LIN {X 0,Y 467.578,Z 154.242,A -85,B 0,C 180,E1 -7774.244,E2 -7774.244} C_VEL
LIN {X 0,Y 467.538,Z 154.245,A -85,B 0,C 180,E1 -7777.188,E2 -7777.188} C_VEL
LIN {X 0,Y 467.566,Z 154.241,A -85,B 0,C 180,E1 -7780.266,E2 -7780.266} C_VEL
LIN {X 0,Y 467.576,Z 154.241,A -85,B 0,C 180,E1 -7782.568,E2 -7782.568} C_VEL
LIN {X 0,Y 467.561,Z 154.246,A -85,B 0,C 180,E1 -7785.055,E2 -7785.055} C_VEL
LIN {X 0,Y 467.579,Z 154.241,A -85,B 0,C 180,E1 -7787.441,E2 -7787.441} C_VEL
LIN {X 0,Y 467.551,Z 154.244,A -85,B 0,C 180,E1 -7790.855,E2 -7790.855} C_VEL
LIN {X 0,Y 467.55,Z 154.243,A -85,B 0,C 180,E1 -7794.263,E2 -7794.263} C_VEL
LIN {X 0,Y 467.576,Z 154.241,A -85,B 0,C 180,E1 -7797.322,E2 -7797.322} C_VEL
LIN {X 0,Y 467.572,Z 154.242,A -85,B 0,C 180,E1 -7800.667,E2 -7800.667} C_VEL
LIN {X 0,Y 467.583,Z 154.244,A -85,B 0,C 180,E1 -7803.199,E2 -7803.199} C_VEL
LIN {X 0,Y 467.585,Z 154.242,A -85,B 0,C 180,E1 -7806.471,E2 -7806.471} C_VEL
LIN {X 0,Y 467.62,Z 154.237,A -85,B 0,C 180,E1 -7809.779,E2 -7809.779} C_VEL
LIN {X 0,Y 467.607,Z 154.238,A -85,B 0,C 180,E1 -7812.508,E2 -7812.508} C_VEL
LIN {X 0,Y 467.6,Z 154.239,A -85,B 0,C 180,E1 -7815.198,E2 -7815.198} C_VEL
LIN {X 0,Y 467.59,Z 154.239,A -85,B 0,C 180,E1 -7815.443,E2 -7815.443} C_VEL
LIN {X 0,Y 466.92,Z 154.324,A -85,B 0,C 180,E1 -7816.162,E2 -7816.162} C_VEL
LIN {X 0,Y 464.077,Z 154.675,A -85,B 0,C 180,E1 -7817.33,E2 -7817.33} C_VEL
LIN {X 0,Y 461.679,Z 154.979,A -85,B 0,C 180,E1 -7818.273,E2 -7818.273} C_VEL
LIN {X 0,Y 460.653,Z 155.102,A -85,B 0,C 180,E1 -7819,E2 -7819} C_VEL
LIN {X 0,Y 460.571,Z 155.112,A -85,B 0,C 180,E1 -7819.247,E2 -7819.247} C_VEL
LIN {X 0,Y 460.721,Z 155.095,A -85,B 0,C 180,E1 -7822.54,E2 -7822.54} C_VEL
LIN {X 0,Y 460.698,Z 155.101,A -85,B 0,C 180,E1 -7824.75,E2 -7824.75} C_VEL
LIN {X 0,Y 460.801,Z 155.085,A -85,B 0,C 180,E1 -7827.379,E2 -7827.379} C_VEL
LIN {X 0,Y 460.821,Z 155.086,A -85,B 0,C 180,E1 -7830.001,E2 -7830.001} C_VEL
LIN {X 0,Y 460.793,Z 155.085,A -85,B 0,C 180,E1 -7832.624,E2 -7832.624} C_VEL
LIN {X 0,Y 460.713,Z 155.097,A -85,B 0,C 180,E1 -7836.131,E2 -7836.131} C_VEL
LIN {X 0,Y 460.63,Z 155.107,A -85,B 0,C 180,E1 -7838.777,E2 -7838.777} C_VEL
LIN {X 0,Y 460.6,Z 155.109,A -85,B 0,C 180,E1 -7842.436,E2 -7842.436} C_VEL
LIN {X 0,Y 460.605,Z 155.109,A -85,B 0,C 180,E1 -7845.999,E2 -7845.999} C_VEL
LIN {X 0,Y 460.573,Z 155.114,A -85,B 0,C 180,E1 -7849.617,E2 -7849.617} C_VEL
LIN {X 0,Y 460.515,Z 155.122,A -85,B 0,C 180,E1 -7852.43,E2 -7852.43} C_VEL
LIN {X 0,Y 460.538,Z 155.116,A -85,B 0,C 180,E1 -7855.794,E2 -7855.794} C_VEL
LIN {X 0,Y 460.525,Z 155.12,A -85,B 0,C 180,E1 -7859.233,E2 -7859.233} C_VEL
LIN {X 0,Y 460.534,Z 155.121,A -85,B 0,C 180,E1 -7862.285,E2 -7862.285} C_VEL
LIN {X 0,Y 460.51,Z 155.123,A -85,B 0,C 180,E1 -7865.447,E2 -7865.447} C_VEL
LIN {X 0,Y 460.495,Z 155.125,A -85,B 0,C 180,E1 -7868.89,E2 -7868.89} C_VEL
LIN {X 0,Y 460.514,Z 155.121,A -85,B 0,C 180,E1 -7871.6,E2 -7871.6} C_VEL
LIN {X 0,Y 460.517,Z 155.121,A -85,B 0,C 180,E1 -7874.59,E2 -7874.59} C_VEL
LIN {X 0,Y 460.528,Z 155.119,A -85,B 0,C 180,E1 -7877.819,E2 -7877.819} C_VEL
LIN {X 0,Y 460.526,Z 155.12,A -85,B 0,C 180,E1 -7880.137,E2 -7880.137} C_VEL
LIN {X 0,Y 460.47,Z 155.126,A -85,B 0,C 180,E1 -7883.47,E2 -7883.47} C_VEL
LIN {X 0,Y 460.529,Z 155.12,A -85,B 0,C 180,E1 -7886.675,E2 -7886.675} C_VEL
LIN {X 0,Y 460.61,Z 155.131,A -85,B 0,C 180,E1 -7887.845,E2 -7887.845} C_VEL
LIN {X 0,Y 461.333,Z 159.923,A -85,B 0,C 180,E1 -7889.82,E2 -7889.82} C_VEL
LIN {X 0,Y 461.056,Z 167.48,A -85,B 0,C 180,E1 -7892.787,E2 -7892.787} C_VEL
LIN {X 0,Y 460.72,Z 176.433,A -85,B 0,C 180,E1 -7896.245,E2 -7896.245} C_VEL
LIN {X 0,Y 460.469,Z 184.873,A -85,B 0,C 180,E1 -7899.449,E2 -7899.449} C_VEL
LIN {X 0,Y 460.238,Z 193.485,A -85,B 0,C 180,E1 -7902.676,E2 -7902.676} C_VEL
LIN {X 0,Y 460.05,Z 202.076,A -85,B 0,C 180,E1 -7905.852,E2 -7905.852} C_VEL
LIN {X 0,Y 459.9,Z 210.667,A -85,B 0,C 180,E1 -7908.988,E2 -7908.988} C_VEL
LIN {X 0,Y 459.815,Z 215.225,A -85,B 0,C 180,E1 -7910.599,E2 -7910.599} C_VEL
LIN {X 0,Y 460.939,Z 225.296,A -85,B 0,C 180,E1 -7911.064,E2 -7911.064} C_VEL
LIN {X 0,Y 461.025,Z 231.865,A -85,B 0,C 180,E1 -7911.452,E2 -7911.452} C_VEL
LIN {X 0,Y 460.704,Z 240.677,A -85,B 0,C 180,E1 -7912.109,E2 -7912.109} C_VEL
LIN {X 0,Y 460.448,Z 249.624,A -85,B 0,C 180,E1 -7912.986,E2 -7912.986} C_VEL
LIN {X 0,Y 460.224,Z 256.55,A -85,B 0,C 180,E1 -7913.864,E2 -7913.864} C_VEL
LIN {X 0,Y 460.116,Z 263.238,A -85,B 0,C 180,E1 -7914.961,E2 -7914.961} C_VEL
LIN {X 0,Y 459.946,Z 268.255,A -85,B 0,C 180,E1 -7916.057,E2 -7916.057} C_VEL
LIN {X 0,Y 459.732,Z 272.503,A -85,B 0,C 180,E1 -7917.371,E2 -7917.371} C_VEL
LIN {X 0,Y 459.652,Z 274.384,A -85,B 0,C 180,E1 -7918.248,E2 -7918.248} C_VEL
LIN {X 0,Y 459.577,Z 275.564,A -85,B 0,C 180,E1 -7919.124,E2 -7919.124} C_VEL
LIN {X 0,Y 459.558,Z 276.065,A -85,B 0,C 180,E1 -7920,E2 -7920} C_VEL
LIN {X 0,Y 459.579,Z 275.892,A -85,B 0,C 180,E1 -7920.876,E2 -7920.876} C_VEL
LIN {X 0,Y 459.655,Z 275.048,A -85,B 0,C 180,E1 -7921.752,E2 -7921.752} C_VEL
LIN {X 0,Y 459.875,Z 272.488,A -85,B 0,C 180,E1 -7923.066,E2 -7923.066} C_VEL
LIN {X 0,Y 460.05,Z 269.86,A -85,B 0,C 180,E1 -7923.942,E2 -7923.942} C_VEL
LIN {X 0,Y 460.191,Z 265.403,A -85,B 0,C 180,E1 -7925.038,E2 -7925.038} C_VEL
LIN {X 0,Y 460.275,Z 259.447,A -85,B 0,C 180,E1 -7926.136,E2 -7926.136} C_VEL
LIN {X 0,Y 460.601,Z 252.231,A -85,B 0,C 180,E1 -7927.147,E2 -7927.147} C_VEL
LIN {X 0,Y 461.059,Z 243.259,A -85,B 0,C 180,E1 -7928.106,E2 -7928.106} C_VEL
LIN {X 0,Y 461.405,Z 235.329,A -85,B 0,C 180,E1 -7928.761,E2 -7928.761} C_VEL
LIN {X 0,Y 461.515,Z 226.898,A -85,B 0,C 180,E1 -7929.311,E2 -7929.311} C_VEL
LIN {X 0,Y 460.127,Z 217.109,A -85,B 0,C 180,E1 -7929.839,E2 -7929.839} C_VEL
LIN {X 0,Y 459.966,Z 215.738,A -85,B 0,C 180,E1 -7929.926,E2 -7929.926} C_VEL
LIN {X 0,Y 460.14,Z 208.06,A -85,B 0,C 180,E1 -7932.795,E2 -7932.795} C_VEL
LIN {X 0,Y 460.413,Z 199.745,A -85,B 0,C 180,E1 -7935.948,E2 -7935.948} C_VEL
LIN {X 0,Y 460.666,Z 192.048,A -85,B 0,C 180,E1 -7938.934,E2 -7938.934} C_VEL
LIN {X 0,Y 460.956,Z 184.495,A -85,B 0,C 180,E1 -7941.934,E2 -7941.934} C_VEL
LIN {X 0,Y 461.333,Z 176.432,A -85,B 0,C 180,E1 -7945.249,E2 -7945.249} C_VEL
LIN {X 0,Y 461.894,Z 169.657,A -85,B 0,C 180,E1 -7948.144,E2 -7948.144} C_VEL
LIN {X 0,Y 462.207,Z 164.213,A -85,B 0,C 180,E1 -7950.623,E2 -7950.623} C_VEL
LIN {X 0,Y 461.444,Z 159.416,A -85,B 0,C 180,E1 -7953.103,E2 -7953.103} C_VEL
LIN {X 0,Y 460.528,Z 155.123,A -85,B 0,C 180,E1 -7955.656,E2 -7955.656} C_VEL
LIN {X 0,Y 460.55,Z 155.12,A -85,B 0,C 180,E1 -7958.897,E2 -7958.897} C_VEL
LIN {X 0,Y 460.529,Z 155.122,A -85,B 0,C 180,E1 -7962.181,E2 -7962.181} C_VEL
LIN {X 0,Y 460.52,Z 155.123,A -85,B 0,C 180,E1 -7965.411,E2 -7965.411} C_VEL
LIN {X 0,Y 460.538,Z 155.12,A -85,B 0,C 180,E1 -7968.397,E2 -7968.397} C_VEL
LIN {X 0,Y 460.532,Z 155.122,A -85,B 0,C 180,E1 -7971.266,E2 -7971.266} C_VEL
LIN {X 0,Y 460.514,Z 155.125,A -85,B 0,C 180,E1 -7974.554,E2 -7974.554} C_VEL
LIN {X 0,Y 460.536,Z 155.127,A -85,B 0,C 180,E1 -7975.256,E2 -7975.256} C_VEL
LIN {X 0,Y 461.79,Z 160.451,A -85,B 0,C 180,E1 -7977.813,E2 -7977.813} C_VEL
LIN {X 0,Y 463.204,Z 167.084,A -85,B 0,C 180,E1 -7980.454,E2 -7980.454} C_VEL
LIN {X 0,Y 463.988,Z 171.493,A -85,B 0,C 180,E1 -7981.993,E2 -7981.993} C_VEL
LIN {X 0,Y 463.796,Z 176.053,A -85,B 0,C 180,E1 -7983.386,E2 -7983.386} C_VEL
LIN {X 0,Y 462.66,Z 186.329,A -85,B 0,C 180,E1 -7986.261,E2 -7986.261} C_VEL
LIN {X 0,Y 461.697,Z 198.798,A -85,B 0,C 180,E1 -7989.505,E2 -7989.505} C_VEL
LIN {X 0,Y 461.026,Z 209.902,A -85,B 0,C 180,E1 -7992.248,E2 -7992.248} C_VEL
LIN {X 0,Y 460.564,Z 220.479,A -85,B 0,C 180,E1 -7994.765,E2 -7994.765} C_VEL
LIN {X 0,Y 462.121,Z 233.34,A -85,B 0,C 180,E1 -7995.17,E2 -7995.17} C_VEL
LIN {X 0,Y 462.47,Z 239.24,A -85,B 0,C 180,E1 -7995.393,E2 -7995.393} C_VEL
LIN {X 0,Y 462.083,Z 251.878,A -85,B 0,C 180,E1 -7995.971,E2 -7995.971} C_VEL
LIN {X 0,Y 461.634,Z 263.462,A -85,B 0,C 180,E1 -7996.686,E2 -7996.686} C_VEL
LIN {X 0,Y 461.188,Z 274.136,A -85,B 0,C 180,E1 -7997.522,E2 -7997.522} C_VEL
LIN {X 0,Y 460.843,Z 283.737,A -85,B 0,C 180,E1 -7998.452,E2 -7998.452} C_VEL
LIN {X 0,Y 460.356,Z 293.826,A -85,B 0,C 180,E1 -7999.665,E2 -7999.665} C_VEL
LIN {X 0,Y 460.039,Z 302.681,A -85,B 0,C 180,E1 -8000.99,E2 -8000.99} C_VEL
LIN {X 0,Y 459.842,Z 309.702,A -85,B 0,C 180,E1 -8002.313,E2 -8002.313} C_VEL
LIN {X 0,Y 459.656,Z 316.123,A -85,B 0,C 180,E1 -8003.855,E2 -8003.855} C_VEL
LIN {X 0,Y 459.628,Z 320.303,A -85,B 0,C 180,E1 -8005.174,E2 -8005.174} C_VEL
LIN {X 0,Y 459.628,Z 323.383,A -85,B 0,C 180,E1 -8006.492,E2 -8006.492} C_VEL
LIN {X 0,Y 459.622,Z 324.86,A -85,B 0,C 180,E1 -8007.369,E2 -8007.369} C_VEL
LIN {X 0,Y 459.601,Z 325.903,A -85,B 0,C 180,E1 -8008.246,E2 -8008.246} C_VEL
LIN {X 0,Y 459.56,Z 326.544,A -85,B 0,C 180,E1 -8009.122,E2 -8009.122} C_VEL
LIN {X 0,Y 459.542,Z 326.768,A -85,B 0,C 180,E1 -8009.999,E2 -8009.999} C_VEL
LIN {X 0,Y 459.63,Z 325.922,A -85,B 0,C 180,E1 -8011.751,E2 -8011.751} C_VEL
LIN {X 0,Y 459.621,Z 324.894,A -85,B 0,C 180,E1 -8012.628,E2 -8012.628} C_VEL
LIN {X 0,Y 459.641,Z 323.396,A -85,B 0,C 180,E1 -8013.505,E2 -8013.505} C_VEL
LIN {X 0,Y 459.623,Z 320.313,A -85,B 0,C 180,E1 -8014.823,E2 -8014.823} C_VEL
LIN {X 0,Y 459.713,Z 315.065,A -85,B 0,C 180,E1 -8016.429,E2 -8016.429} C_VEL
LIN {X 0,Y 459.866,Z 308.616,A -85,B 0,C 180,E1 -8017.904,E2 -8017.904} C_VEL
LIN {X 0,Y 460.097,Z 301.234,A -85,B 0,C 180,E1 -8019.228,E2 -8019.228} C_VEL
LIN {X 0,Y 460.348,Z 293.675,A -85,B 0,C 180,E1 -8020.332,E2 -8020.332} C_VEL
LIN {X 0,Y 460.797,Z 284.488,A -85,B 0,C 180,E1 -8021.434,E2 -8021.434} C_VEL
LIN {X 0,Y 461.196,Z 274.181,A -85,B 0,C 180,E1 -8022.43,E2 -8022.43} C_VEL
LIN {X 0,Y 461.628,Z 262.754,A -85,B 0,C 180,E1 -8023.311,E2 -8023.311} C_VEL
LIN {X 0,Y 462.054,Z 250.719,A -85,B 0,C 180,E1 -8024.027,E2 -8024.027} C_VEL
LIN {X 0,Y 462.432,Z 237.387,A -85,B 0,C 180,E1 -8024.606,E2 -8024.606} C_VEL
LIN {X 0,Y 460.969,Z 224.354,A -85,B 0,C 180,E1 -8025.02,E2 -8025.02} C_VEL
LIN {X 0,Y 460.482,Z 220.513,A -85,B 0,C 180,E1 -8025.121,E2 -8025.121} C_VEL
LIN {X 0,Y 461.162,Z 205.323,A -85,B 0,C 180,E1 -8028.663,E2 -8028.663} C_VEL
LIN {X 0,Y 461.925,Z 189.777,A -85,B 0,C 180,E1 -8032.354,E2 -8032.354} C_VEL
LIN {X 0,Y 462.774,Z 176.253,A -85,B 0,C 180,E1 -8035.645,E2 -8035.645} C_VEL
LIN {X 0,Y 463.153,Z 170.459,A -85,B 0,C 180,E1 -8037.078,E2 -8037.078} C_VEL
LIN {X 0,Y 462.725,Z 165.962,A -85,B 0,C 180,E1 -8038.246,E2 -8038.246} C_VEL
LIN {X 0,Y 460.54,Z 155.121,A -85,B 0,C 180,E1 -8041.227,E2 -8041.227} C_VEL
LIN {X 0,Y 460.529,Z 155.122,A -85,B 0,C 180,E1 -8044.504,E2 -8044.504} C_VEL
LIN {X 0,Y 460.521,Z 155.121,A -85,B 0,C 180,E1 -8047.619,E2 -8047.619} C_VEL
LIN {X 0,Y 460.518,Z 155.121,A -85,B 0,C 180,E1 -8051.01,E2 -8051.01} C_VEL
LIN {X 0,Y 460.506,Z 155.123,A -85,B 0,C 180,E1 -8054.587,E2 -8054.587} C_VEL
LIN {X 0,Y 460.538,Z 155.12,A -85,B 0,C 180,E1 -8057.82,E2 -8057.82} C_VEL
LIN {X 0,Y 460.557,Z 155.116,A -85,B 0,C 180,E1 -8061.097,E2 -8061.097} C_VEL
LIN {X 0,Y 460.496,Z 155.123,A -85,B 0,C 180,E1 -8064.553,E2 -8064.553} C_VEL
LIN {X 0,Y 460.521,Z 155.123,A -85,B 0,C 180,E1 -8067.715,E2 -8067.715} C_VEL
LIN {X 0,Y 460.535,Z 155.12,A -85,B 0,C 180,E1 -8070.769,E2 -8070.769} C_VEL
LIN {X 0,Y 460.551,Z 155.117,A -85,B 0,C 180,E1 -8073.734,E2 -8073.734} C_VEL
LIN {X 0,Y 460.531,Z 155.117,A -85,B 0,C 180,E1 -8076.623,E2 -8076.623} C_VEL
LIN {X 0,Y 460.537,Z 155.122,A -85,B 0,C 180,E1 -8079.452,E2 -8079.452} C_VEL
LIN {X 0,Y 460.546,Z 155.118,A -85,B 0,C 180,E1 -8082.229,E2 -8082.229} C_VEL
LIN {X 0,Y 460.551,Z 155.117,A -85,B 0,C 180,E1 -8084.964,E2 -8084.964} C_VEL
LIN {X 0,Y 460.613,Z 155.112,A -85,B 0,C 180,E1 -8087.666,E2 -8087.666} C_VEL
LIN {X 0,Y 460.611,Z 155.112,A -85,B 0,C 180,E1 -8091.223,E2 -8091.223} C_VEL
LIN {X 0,Y 460.698,Z 155.098,A -85,B 0,C 180,E1 -8093.87,E2 -8093.87} C_VEL
LIN {X 0,Y 460.812,Z 155.086,A -85,B 0,C 180,E1 -8097.378,E2 -8097.378} C_VEL
LIN {X 0,Y 460.836,Z 155.081,A -85,B 0,C 180,E1 -8100,E2 -8100} C_VEL
LIN {X 0,Y 460.78,Z 155.089,A -85,B 0,C 180,E1 -8102.623,E2 -8102.623} C_VEL
LIN {X 0,Y 460.694,Z 155.1,A -85,B 0,C 180,E1 -8106.13,E2 -8106.13} C_VEL
LIN {X 0,Y 460.615,Z 155.109,A -85,B 0,C 180,E1 -8108.776,E2 -8108.776} C_VEL
LIN {X 0,Y 460.619,Z 155.109,A -85,B 0,C 180,E1 -8112.457,E2 -8112.457} C_VEL
LIN {X 0,Y 460.585,Z 155.112,A -85,B 0,C 180,E1 -8115.998,E2 -8115.998} C_VEL
LIN {X 0,Y 460.557,Z 155.116,A -85,B 0,C 180,E1 -8118.903,E2 -8118.903} C_VEL
LIN {X 0,Y 460.549,Z 155.118,A -85,B 0,C 180,E1 -8121.484,E2 -8121.484} C_VEL
LIN {X 0,Y 460.524,Z 155.122,A -85,B 0,C 180,E1 -8124.333,E2 -8124.333} C_VEL
LIN {X 0,Y 460.521,Z 155.118,A -85,B 0,C 180,E1 -8127.247,E2 -8127.247} C_VEL
LIN {X 0,Y 460.496,Z 155.123,A -85,B 0,C 180,E1 -8130.241,E2 -8130.241} C_VEL
LIN {X 0,Y 460.517,Z 155.123,A -85,B 0,C 180,E1 -8133.326,E2 -8133.326} C_VEL
LIN {X 0,Y 460.467,Z 155.128,A -85,B 0,C 180,E1 -8136.53,E2 -8136.53} C_VEL
LIN {X 0,Y 460.546,Z 155.119,A -85,B 0,C 180,E1 -8139.861,E2 -8139.861} C_VEL
LIN {X 0,Y 460.506,Z 155.122,A -85,B 0,C 180,E1 -8142.902,E2 -8142.902} C_VEL
LIN {X 0,Y 460.51,Z 155.122,A -85,B 0,C 180,E1 -8145.831,E2 -8145.831} C_VEL
LIN {X 0,Y 460.524,Z 155.12,A -85,B 0,C 180,E1 -8148.99,E2 -8148.99} C_VEL
LIN {X 0,Y 460.51,Z 155.124,A -85,B 0,C 180,E1 -8151.268,E2 -8151.268} C_VEL
LIN {X 0,Y 460.501,Z 155.122,A -85,B 0,C 180,E1 -8154.556,E2 -8154.556} C_VEL
LIN {X 0,Y 460.527,Z 155.12,A -85,B 0,C 180,E1 -8157.717,E2 -8157.717} C_VEL
LIN {X 0,Y 460.541,Z 155.118,A -85,B 0,C 180,E1 -8160.771,E2 -8160.771} C_VEL
LIN {X 0,Y 460.537,Z 155.117,A -85,B 0,C 180,E1 -8163.735,E2 -8163.735} C_VEL
LIN {X 0,Y 460.539,Z 155.121,A -85,B 0,C 180,E1 -8166.625,E2 -8166.625} C_VEL
LIN {X 0,Y 460.548,Z 155.117,A -85,B 0,C 180,E1 -8169.454,E2 -8169.454} C_VEL
LIN {X 0,Y 460.557,Z 155.116,A -85,B 0,C 180,E1 -8172.232,E2 -8172.232} C_VEL
LIN {X 0,Y 460.56,Z 155.117,A -85,B 0,C 180,E1 -8174.966,E2 -8174.966} C_VEL
LIN {X 0,Y 460.608,Z 155.111,A -85,B 0,C 180,E1 -8178.561,E2 -8178.561} C_VEL
LIN {X 0,Y 460.571,Z 155.112,A -85,B 0,C 180,E1 -8179.247,E2 -8179.247} C_VEL
LIN {X 0,Y 459.917,Z 155.198,A -85,B 0,C 180,E1 -8179.977,E2 -8179.977} C_VEL
LIN {X 0,Y 457.101,Z 155.547,A -85,B 0,C 180,E1 -8181.164,E2 -8181.164} C_VEL
LIN {X 0,Y 454.725,Z 155.844,A -85,B 0,C 180,E1 -8182.121,E2 -8182.121} C_VEL
LIN {X 0,Y 453.715,Z 155.969,A -85,B 0,C 180,E1 -8182.86,E2 -8182.86} C_VEL
LIN {X 0,Y 453.638,Z 155.978,A -85,B 0,C 180,E1 -8183.11,E2 -8183.11} C_VEL
LIN {X 0,Y 453.672,Z 155.975,A -85,B 0,C 180,E1 -8184.668,E2 -8184.668} C_VEL
LIN {X 0,Y 453.746,Z 155.964,A -85,B 0,C 180,E1 -8187.338,E2 -8187.338} C_VEL
LIN {X 0,Y 453.79,Z 155.962,A -85,B 0,C 180,E1 -8190.001,E2 -8190.001} C_VEL
LIN {X 0,Y 453.737,Z 155.964,A -85,B 0,C 180,E1 -8192.665,E2 -8192.665} C_VEL
LIN {X 0,Y 453.68,Z 155.973,A -85,B 0,C 180,E1 -8196.227,E2 -8196.227} C_VEL
LIN {X 0,Y 453.594,Z 155.984,A -85,B 0,C 180,E1 -8198.915,E2 -8198.915} C_VEL
LIN {X 0,Y 453.567,Z 155.985,A -85,B 0,C 180,E1 -8202.53,E2 -8202.53} C_VEL
LIN {X 0,Y 453.549,Z 155.988,A -85,B 0,C 180,E1 -8206.197,E2 -8206.197} C_VEL
LIN {X 0,Y 453.522,Z 155.994,A -85,B 0,C 180,E1 -8209.041,E2 -8209.041} C_VEL
LIN {X 0,Y 453.481,Z 155.999,A -85,B 0,C 180,E1 -8211.837,E2 -8211.837} C_VEL
LIN {X 0,Y 453.473,Z 155.997,A -85,B 0,C 180,E1 -8214.738,E2 -8214.738} C_VEL
LIN {X 0,Y 453.467,Z 155.998,A -85,B 0,C 180,E1 -8217.944,E2 -8217.944} C_VEL
LIN {X 0,Y 453.479,Z 155.999,A -85,B 0,C 180,E1 -8220.761,E2 -8220.761} C_VEL
LIN {X 0,Y 453.473,Z 155.999,A -85,B 0,C 180,E1 -8223.914,E2 -8223.914} C_VEL
LIN {X 0,Y 453.443,Z 156.003,A -85,B 0,C 180,E1 -8227.192,E2 -8227.192} C_VEL
LIN {X 0,Y 453.475,Z 156,A -85,B 0,C 180,E1 -8230.612,E2 -8230.612} C_VEL
LIN {X 0,Y 453.465,Z 156.001,A -85,B 0,C 180,E1 -8234.222,E2 -8234.222} C_VEL
LIN {X 0,Y 453.467,Z 156.001,A -85,B 0,C 180,E1 -8237.005,E2 -8237.005} C_VEL
LIN {X 0,Y 453.499,Z 155.994,A -85,B 0,C 180,E1 -8239.41,E2 -8239.41} C_VEL
LIN {X 0,Y 453.444,Z 156.001,A -85,B 0,C 180,E1 -8242.809,E2 -8242.809} C_VEL
LIN {X 0,Y 453.475,Z 155.999,A -85,B 0,C 180,E1 -8246.087,E2 -8246.087} C_VEL
LIN {X 0,Y 453.588,Z 156.076,A -85,B 0,C 180,E1 -8247.752,E2 -8247.752} C_VEL
LIN {X 0,Y 454.308,Z 161.581,A -85,B 0,C 180,E1 -8250.033,E2 -8250.033} C_VEL
LIN {X 0,Y 453.974,Z 169.864,A -85,B 0,C 180,E1 -8253.324,E2 -8253.324} C_VEL
LIN {X 0,Y 453.622,Z 178.6,A -85,B 0,C 180,E1 -8256.729,E2 -8256.729} C_VEL
LIN {X 0,Y 453.381,Z 187.277,A -85,B 0,C 180,E1 -8260.06,E2 -8260.06} C_VEL
LIN {X 0,Y 453.168,Z 195.94,A -85,B 0,C 180,E1 -8263.327,E2 -8263.327} C_VEL
LIN {X 0,Y 452.947,Z 204.557,A -85,B 0,C 180,E1 -8266.541,E2 -8266.541} C_VEL
LIN {X 0,Y 452.762,Z 213.16,A -85,B 0,C 180,E1 -8269.717,E2 -8269.717} C_VEL
LIN {X 0,Y 452.753,Z 215.324,A -85,B 0,C 180,E1 -8270.451,E2 -8270.451} C_VEL
LIN {X 0,Y 453.895,Z 225.363,A -85,B 0,C 180,E1 -8270.924,E2 -8270.924} C_VEL
LIN {X 0,Y 454.018,Z 231.934,A -85,B 0,C 180,E1 -8271.319,E2 -8271.319} C_VEL
LIN {X 0,Y 453.675,Z 240.772,A -85,B 0,C 180,E1 -8271.986,E2 -8271.986} C_VEL
LIN {X 0,Y 453.405,Z 249.758,A -85,B 0,C 180,E1 -8272.877,E2 -8272.877} C_VEL
LIN {X 0,Y 453.184,Z 256.726,A -85,B 0,C 180,E1 -8273.768,E2 -8273.768} C_VEL
LIN {X 0,Y 453.038,Z 263.457,A -85,B 0,C 180,E1 -8274.882,E2 -8274.882} C_VEL
LIN {X 0,Y 452.88,Z 268.517,A -85,B 0,C 180,E1 -8275.996,E2 -8275.996} C_VEL
LIN {X 0,Y 452.656,Z 272.809,A -85,B 0,C 180,E1 -8277.33,E2 -8277.33} C_VEL
LIN {X 0,Y 452.576,Z 274.721,A -85,B 0,C 180,E1 -8278.22,E2 -8278.22} C_VEL
LIN {X 0,Y 452.512,Z 275.932,A -85,B 0,C 180,E1 -8279.11,E2 -8279.11} C_VEL
LIN {X 0,Y 452.491,Z 276.463,A -85,B 0,C 180,E1 -8280,E2 -8280} C_VEL
LIN {X 0,Y 452.513,Z 276.322,A -85,B 0,C 180,E1 -8280.89,E2 -8280.89} C_VEL
LIN {X 0,Y 452.596,Z 275.507,A -85,B 0,C 180,E1 -8281.78,E2 -8281.78} C_VEL
LIN {X 0,Y 452.828,Z 272.992,A -85,B 0,C 180,E1 -8283.114,E2 -8283.114} C_VEL
LIN {X 0,Y 453.005,Z 270.405,A -85,B 0,C 180,E1 -8284.003,E2 -8284.003} C_VEL
LIN {X 0,Y 453.159,Z 266.01,A -85,B 0,C 180,E1 -8285.116,E2 -8285.116} C_VEL
LIN {X 0,Y 453.254,Z 260.142,A -85,B 0,C 180,E1 -8286.231,E2 -8286.231} C_VEL
LIN {X 0,Y 453.627,Z 253.039,A -85,B 0,C 180,E1 -8287.257,E2 -8287.257} C_VEL
LIN {X 0,Y 454.099,Z 244.254,A -85,B 0,C 180,E1 -8288.231,E2 -8288.231} C_VEL
LIN {X 0,Y 454.541,Z 235.084,A -85,B 0,C 180,E1 -8289.007,E2 -8289.007} C_VEL
LIN {X 0,Y 454.536,Z 226.624,A -85,B 0,C 180,E1 -8289.568,E2 -8289.568} C_VEL
LIN {X 0,Y 452.893,Z 215.887,A -85,B 0,C 180,E1 -8290.167,E2 -8290.167} C_VEL
LIN {X 0,Y 453.11,Z 208.424,A -85,B 0,C 180,E1 -8292.997,E2 -8292.997} C_VEL
LIN {X 0,Y 453.415,Z 200.124,A -85,B 0,C 180,E1 -8296.201,E2 -8296.201} C_VEL
LIN {X 0,Y 453.711,Z 192.031,A -85,B 0,C 180,E1 -8299.406,E2 -8299.406} C_VEL
LIN {X 0,Y 453.987,Z 184.947,A -85,B 0,C 180,E1 -8302.289,E2 -8302.289} C_VEL
LIN {X 0,Y 454.387,Z 178.087,A -85,B 0,C 180,E1 -8305.172,E2 -8305.172} C_VEL
LIN {X 0,Y 455.015,Z 170.966,A -85,B 0,C 180,E1 -8308.308,E2 -8308.308} C_VEL
LIN {X 0,Y 455.326,Z 165.982,A -85,B 0,C 180,E1 -8310.621,E2 -8310.621} C_VEL
LIN {X 0,Y 454.732,Z 161.992,A -85,B 0,C 180,E1 -8312.747,E2 -8312.747} C_VEL
LIN {X 0,Y 453.987,Z 158.278,A -85,B 0,C 180,E1 -8314.945,E2 -8314.945} C_VEL
LIN {X 0,Y 453.45,Z 156.005,A -85,B 0,C 180,E1 -8316.583,E2 -8316.583} C_VEL
LIN {X 0,Y 453.496,Z 155.999,A -85,B 0,C 180,E1 -8319.449,E2 -8319.449} C_VEL
LIN {X 0,Y 453.482,Z 155.999,A -85,B 0,C 180,E1 -8321.934,E2 -8321.934} C_VEL
LIN {X 0,Y 453.491,Z 155.998,A -85,B 0,C 180,E1 -8325.471,E2 -8325.471} C_VEL
LIN {X 0,Y 453.485,Z 155.999,A -85,B 0,C 180,E1 -8328.209,E2 -8328.209} C_VEL
LIN {X 0,Y 453.5,Z 155.998,A -85,B 0,C 180,E1 -8330.793,E2 -8330.793} C_VEL
LIN {X 0,Y 453.478,Z 156.021,A -85,B 0,C 180,E1 -8334.329,E2 -8334.329} C_VEL
LIN {X 0,Y 454.505,Z 160.218,A -85,B 0,C 180,E1 -8336.616,E2 -8336.616} C_VEL
LIN {X 0,Y 455.912,Z 166.574,A -85,B 0,C 180,E1 -8339.421,E2 -8339.421} C_VEL
LIN {X 0,Y 457.004,Z 172.24,A -85,B 0,C 180,E1 -8341.527,E2 -8341.527} C_VEL
LIN {X 0,Y 457.184,Z 175.23,A -85,B 0,C 180,E1 -8342.536,E2 -8342.536} C_VEL
LIN {X 0,Y 456.05,Z 185.023,A -85,B 0,C 180,E1 -8345.411,E2 -8345.411} C_VEL
LIN {X 0,Y 454.888,Z 197.193,A -85,B 0,C 180,E1 -8348.71,E2 -8348.71} C_VEL
LIN {X 0,Y 454.07,Z 209.97,A -85,B 0,C 180,E1 -8351.966,E2 -8351.966} C_VEL
LIN {X 0,Y 453.56,Z 220.544,A -85,B 0,C 180,E1 -8354.537,E2 -8354.537} C_VEL
LIN {X 0,Y 455.114,Z 232.788,A -85,B 0,C 180,E1 -8354.922,E2 -8354.922} C_VEL
LIN {X 0,Y 455.569,Z 239.804,A -85,B 0,C 180,E1 -8355.195,E2 -8355.195} C_VEL
LIN {X 0,Y 455.183,Z 251.645,A -85,B 0,C 180,E1 -8355.753,E2 -8355.753} C_VEL
LIN {X 0,Y 454.706,Z 263.183,A -85,B 0,C 180,E1 -8356.479,E2 -8356.479} C_VEL
LIN {X 0,Y 454.186,Z 274.366,A -85,B 0,C 180,E1 -8357.374,E2 -8357.374} C_VEL
LIN {X 0,Y 453.805,Z 284.42,A -85,B 0,C 180,E1 -8358.384,E2 -8358.384} C_VEL
LIN {X 0,Y 453.34,Z 293.498,A -85,B 0,C 180,E1 -8359.503,E2 -8359.503} C_VEL
LIN {X 0,Y 452.993,Z 302.337,A -85,B 0,C 180,E1 -8360.848,E2 -8360.848} C_VEL
LIN {X 0,Y 452.757,Z 309.345,A -85,B 0,C 180,E1 -8362.192,E2 -8362.192} C_VEL
LIN {X 0,Y 452.585,Z 315.769,A -85,B 0,C 180,E1 -8363.758,E2 -8363.758} C_VEL
LIN {X 0,Y 452.558,Z 319.943,A -85,B 0,C 180,E1 -8365.099,E2 -8365.099} C_VEL
LIN {X 0,Y 452.525,Z 323.013,A -85,B 0,C 180,E1 -8366.437,E2 -8366.437} C_VEL
LIN {X 0,Y 452.544,Z 324.483,A -85,B 0,C 180,E1 -8367.328,E2 -8367.328} C_VEL
LIN {X 0,Y 452.511,Z 325.521,A -85,B 0,C 180,E1 -8368.219,E2 -8368.219} C_VEL
LIN {X 0,Y 452.495,Z 326.159,A -85,B 0,C 180,E1 -8369.109,E2 -8369.109} C_VEL
LIN {X 0,Y 452.475,Z 326.369,A -85,B 0,C 180,E1 -8369.999,E2 -8369.999} C_VEL
LIN {X 0,Y 452.495,Z 326.137,A -85,B 0,C 180,E1 -8370.889,E2 -8370.889} C_VEL
LIN {X 0,Y 452.538,Z 325.507,A -85,B 0,C 180,E1 -8371.778,E2 -8371.778} C_VEL
LIN {X 0,Y 452.544,Z 324.467,A -85,B 0,C 180,E1 -8372.669,E2 -8372.669} C_VEL
LIN {X 0,Y 452.539,Z 322.948,A -85,B 0,C 180,E1 -8373.56,E2 -8373.56} C_VEL
LIN {X 0,Y 452.554,Z 319.839,A -85,B 0,C 180,E1 -8374.898,E2 -8374.898} C_VEL
LIN {X 0,Y 452.609,Z 315.05,A -85,B 0,C 180,E1 -8376.394,E2 -8376.394} C_VEL
LIN {X 0,Y 452.756,Z 309.145,A -85,B 0,C 180,E1 -8377.805,E2 -8377.805} C_VEL
LIN {X 0,Y 453.002,Z 301.97,A -85,B 0,C 180,E1 -8379.149,E2 -8379.149} C_VEL
LIN {X 0,Y 453.315,Z 292.978,A -85,B 0,C 180,E1 -8380.494,E2 -8380.494} C_VEL
LIN {X 0,Y 453.788,Z 283.674,A -85,B 0,C 180,E1 -8381.614,E2 -8381.614} C_VEL
LIN {X 0,Y 454.203,Z 273.105,A -85,B 0,C 180,E1 -8382.635,E2 -8382.635} C_VEL
LIN {X 0,Y 454.683,Z 261.654,A -85,B 0,C 180,E1 -8383.518,E2 -8383.518} C_VEL
LIN {X 0,Y 455.091,Z 249.255,A -85,B 0,C 180,E1 -8384.247,E2 -8384.247} C_VEL
LIN {X 0,Y 455.333,Z 236.604,A -85,B 0,C 180,E1 -8384.796,E2 -8384.796} C_VEL
LIN {X 0,Y 453.906,Z 224.212,A -85,B 0,C 180,E1 -8385.191,E2 -8385.191} C_VEL
LIN {X 0,Y 453.46,Z 220.471,A -85,B 0,C 180,E1 -8385.302,E2 -8385.302} C_VEL
LIN {X 0,Y 454.068,Z 206.965,A -85,B 0,C 180,E1 -8388.498,E2 -8388.498} C_VEL
LIN {X 0,Y 454.832,Z 192.43,A -85,B 0,C 180,E1 -8392.011,E2 -8392.011} C_VEL
LIN {X 0,Y 455.772,Z 177.986,A -85,B 0,C 180,E1 -8395.577,E2 -8395.577} C_VEL
LIN {X 0,Y 456.175,Z 170.268,A -85,B 0,C 180,E1 -8397.527,E2 -8397.527} C_VEL
LIN {X 0,Y 454.541,Z 161.142,A -85,B 0,C 180,E1 -8400.019,E2 -8400.019} C_VEL
LIN {X 0,Y 453.46,Z 156.002,A -85,B 0,C 180,E1 -8401.523,E2 -8401.523} C_VEL
LIN {X 0,Y 453.483,Z 155.998,A -85,B 0,C 180,E1 -8404.776,E2 -8404.776} C_VEL
LIN {X 0,Y 453.46,Z 156,A -85,B 0,C 180,E1 -8408.31,E2 -8408.31} C_VEL
LIN {X 0,Y 453.485,Z 155.999,A -85,B 0,C 180,E1 -8410.607,E2 -8410.607} C_VEL
LIN {X 0,Y 453.454,Z 156.003,A -85,B 0,C 180,E1 -8414.22,E2 -8414.22} C_VEL
LIN {X 0,Y 453.483,Z 155.998,A -85,B 0,C 180,E1 -8417.007,E2 -8417.007} C_VEL
LIN {X 0,Y 453.522,Z 155.994,A -85,B 0,C 180,E1 -8420.553,E2 -8420.553} C_VEL
LIN {X 0,Y 453.439,Z 156.003,A -85,B 0,C 180,E1 -8423.916,E2 -8423.916} C_VEL
LIN {X 0,Y 453.471,Z 155.998,A -85,B 0,C 180,E1 -8427.15,E2 -8427.15} C_VEL
LIN {X 0,Y 453.502,Z 155.995,A -85,B 0,C 180,E1 -8430.27,E2 -8430.27} C_VEL
LIN {X 0,Y 453.499,Z 155.995,A -85,B 0,C 180,E1 -8433.293,E2 -8433.293} C_VEL
LIN {X 0,Y 453.487,Z 155.996,A -85,B 0,C 180,E1 -8436.238,E2 -8436.238} C_VEL
LIN {X 0,Y 453.468,Z 155.999,A -85,B 0,C 180,E1 -8439.117,E2 -8439.117} C_VEL
LIN {X 0,Y 453.498,Z 155.995,A -85,B 0,C 180,E1 -8441.944,E2 -8441.944} C_VEL
LIN {X 0,Y 453.525,Z 155.993,A -85,B 0,C 180,E1 -8444.726,E2 -8444.726} C_VEL
LIN {X 0,Y 453.587,Z 155.986,A -85,B 0,C 180,E1 -8447.472,E2 -8447.472} C_VEL
LIN {X 0,Y 453.574,Z 155.988,A -85,B 0,C 180,E1 -8451.086,E2 -8451.086} C_VEL
LIN {X 0,Y 453.665,Z 155.974,A -85,B 0,C 180,E1 -8453.774,E2 -8453.774} C_VEL
LIN {X 0,Y 453.753,Z 155.965,A -85,B 0,C 180,E1 -8457.337,E2 -8457.337} C_VEL
LIN {X 0,Y 453.806,Z 155.956,A -85,B 0,C 180,E1 -8460,E2 -8460} C_VEL
LIN {X 0,Y 453.724,Z 155.968,A -85,B 0,C 180,E1 -8462.663,E2 -8462.663} C_VEL
LIN {X 0,Y 453.662,Z 155.976,A -85,B 0,C 180,E1 -8466.225,E2 -8466.225} C_VEL
LIN {X 0,Y 453.579,Z 155.986,A -85,B 0,C 180,E1 -8468.914,E2 -8468.914} C_VEL
LIN {X 0,Y 453.587,Z 155.985,A -85,B 0,C 180,E1 -8472.551,E2 -8472.551} C_VEL
LIN {X 0,Y 453.53,Z 155.993,A -85,B 0,C 180,E1 -8476.196,E2 -8476.196} C_VEL
LIN {X 0,Y 453.506,Z 155.994,A -85,B 0,C 180,E1 -8479.042,E2 -8479.042} C_VEL
LIN {X 0,Y 453.487,Z 155.997,A -85,B 0,C 180,E1 -8481.836,E2 -8481.836} C_VEL
LIN {X 0,Y 453.492,Z 155.997,A -85,B 0,C 180,E1 -8484.736,E2 -8484.736} C_VEL
LIN {X 0,Y 453.492,Z 155.999,A -85,B 0,C 180,E1 -8487.954,E2 -8487.954} C_VEL
LIN {X 0,Y 453.462,Z 155.999,A -85,B 0,C 180,E1 -8490.761,E2 -8490.761} C_VEL
LIN {X 0,Y 453.466,Z 155.999,A -85,B 0,C 180,E1 -8493.914,E2 -8493.914} C_VEL
LIN {X 0,Y 453.459,Z 155.999,A -85,B 0,C 180,E1 -8497.189,E2 -8497.189} C_VEL
LIN {X 0,Y 453.505,Z 155.995,A -85,B 0,C 180,E1 -8499.448,E2 -8499.448} C_VEL
LIN {X 0,Y 453.457,Z 156.001,A -85,B 0,C 180,E1 -8502.996,E2 -8502.996} C_VEL
LIN {X 0,Y 453.464,Z 156,A -85,B 0,C 180,E1 -8505.781,E2 -8505.781} C_VEL
LIN {X 0,Y 453.473,Z 155.999,A -85,B 0,C 180,E1 -8508.211,E2 -8508.211} C_VEL
LIN {X 0,Y 453.478,Z 155.997,A -85,B 0,C 180,E1 -8510.796,E2 -8510.796} C_VEL
LIN {X 0,Y 453.445,Z 156,A -85,B 0,C 180,E1 -8513.919,E2 -8513.919} C_VEL
LIN {X 0,Y 453.477,Z 155.998,A -85,B 0,C 180,E1 -8517.153,E2 -8517.153} C_VEL
LIN {X 0,Y 453.509,Z 155.995,A -85,B 0,C 180,E1 -8520.273,E2 -8520.273} C_VEL
LIN {X 0,Y 453.484,Z 155.999,A -85,B 0,C 180,E1 -8523.294,E2 -8523.294} C_VEL
LIN {X 0,Y 453.488,Z 155.995,A -85,B 0,C 180,E1 -8526.24,E2 -8526.24} C_VEL
LIN {X 0,Y 453.479,Z 155.997,A -85,B 0,C 180,E1 -8529.119,E2 -8529.119} C_VEL
LIN {X 0,Y 453.51,Z 155.995,A -85,B 0,C 180,E1 -8531.946,E2 -8531.946} C_VEL
LIN {X 0,Y 453.536,Z 155.993,A -85,B 0,C 180,E1 -8534.728,E2 -8534.728} C_VEL
LIN {X 0,Y 453.557,Z 155.992,A -85,B 0,C 180,E1 -8538.38,E2 -8538.38} C_VEL
LIN {X 0,Y 453.652,Z 155.979,A -85,B 0,C 180,E1 -8541.987,E2 -8541.987} C_VEL
LIN {X 0,Y 453.638,Z 155.978,A -85,B 0,C 180,E1 -8543.11,E2 -8543.11} C_VEL
LIN {X 0,Y 452.955,Z 156.064,A -85,B 0,C 180,E1 -8543.85,E2 -8543.85} C_VEL
LIN {X 0,Y 450.009,Z 156.43,A -85,B 0,C 180,E1 -8545.052,E2 -8545.052} C_VEL
LIN {X 0,Y 447.583,Z 156.732,A -85,B 0,C 180,E1 -8546.021,E2 -8546.021} C_VEL
LIN {X 0,Y 446.64,Z 156.85,A -85,B 0,C 180,E1 -8546.772,E2 -8546.772} C_VEL
LIN {X 0,Y 446.617,Z 156.852,A -85,B 0,C 180,E1 -8547.025,E2 -8547.025} C_VEL
LIN {X 0,Y 446.739,Z 156.84,A -85,B 0,C 180,E1 -8550.001,E2 -8550.001} C_VEL
LIN {X 0,Y 446.684,Z 156.843,A -85,B 0,C 180,E1 -8552.707,E2 -8552.707} C_VEL
LIN {X 0,Y 446.65,Z 156.849,A -85,B 0,C 180,E1 -8556.325,E2 -8556.325} C_VEL
LIN {X 0,Y 446.54,Z 156.863,A -85,B 0,C 180,E1 -8559.057,E2 -8559.057} C_VEL
LIN {X 0,Y 446.525,Z 156.862,A -85,B 0,C 180,E1 -8562.731,E2 -8562.731} C_VEL
LIN {X 0,Y 446.493,Z 156.867,A -85,B 0,C 180,E1 -8566.46,E2 -8566.46} C_VEL
LIN {X 0,Y 446.473,Z 156.871,A -85,B 0,C 180,E1 -8569.304,E2 -8569.304} C_VEL
LIN {X 0,Y 446.422,Z 156.877,A -85,B 0,C 180,E1 -8572.201,E2 -8572.201} C_VEL
LIN {X 0,Y 446.425,Z 156.879,A -85,B 0,C 180,E1 -8575.155,E2 -8575.155} C_VEL
LIN {X 0,Y 446.441,Z 156.873,A -85,B 0,C 180,E1 -8578.183,E2 -8578.183} C_VEL
LIN {X 0,Y 446.419,Z 156.877,A -85,B 0,C 180,E1 -8581.301,E2 -8581.301} C_VEL
LIN {X 0,Y 446.427,Z 156.876,A -85,B 0,C 180,E1 -8584.524,E2 -8584.524} C_VEL
LIN {X 0,Y 446.402,Z 156.877,A -85,B 0,C 180,E1 -8588.077,E2 -8588.077} C_VEL
LIN {X 0,Y 446.411,Z 156.877,A -85,B 0,C 180,E1 -8591.394,E2 -8591.394} C_VEL
LIN {X 0,Y 446.456,Z 156.874,A -85,B 0,C 180,E1 -8595.104,E2 -8595.104} C_VEL
LIN {X 0,Y 446.433,Z 156.879,A -85,B 0,C 180,E1 -8598.609,E2 -8598.609} C_VEL
LIN {X 0,Y 446.405,Z 156.879,A -85,B 0,C 180,E1 -8601.924,E2 -8601.924} C_VEL
LIN {X 0,Y 446.428,Z 156.878,A -85,B 0,C 180,E1 -8605.477,E2 -8605.477} C_VEL
LIN {X 0,Y 446.538,Z 157.009,A -85,B 0,C 180,E1 -8607.648,E2 -8607.648} C_VEL
LIN {X 0,Y 447.248,Z 162.143,A -85,B 0,C 180,E1 -8609.812,E2 -8609.812} C_VEL
LIN {X 0,Y 446.998,Z 169.746,A -85,B 0,C 180,E1 -8612.873,E2 -8612.873} C_VEL
LIN {X 0,Y 446.635,Z 178.537,A -85,B 0,C 180,E1 -8616.35,E2 -8616.35} C_VEL
LIN {X 0,Y 446.338,Z 187.247,A -85,B 0,C 180,E1 -8619.732,E2 -8619.732} C_VEL
LIN {X 0,Y 446.114,Z 195.915,A -85,B 0,C 180,E1 -8623.055,E2 -8623.055} C_VEL
LIN {X 0,Y 445.886,Z 204.555,A -85,B 0,C 180,E1 -8626.324,E2 -8626.324} C_VEL
LIN {X 0,Y 445.702,Z 213.217,A -85,B 0,C 180,E1 -8629.552,E2 -8629.552} C_VEL
LIN {X 0,Y 445.65,Z 215.234,A -85,B 0,C 180,E1 -8630.297,E2 -8630.297} C_VEL
LIN {X 0,Y 446.916,Z 226.351,A -85,B 0,C 180,E1 -8630.838,E2 -8630.838} C_VEL
LIN {X 0,Y 446.931,Z 233.588,A -85,B 0,C 180,E1 -8631.295,E2 -8631.295} C_VEL
LIN {X 0,Y 446.562,Z 243.536,A -85,B 0,C 180,E1 -8632.108,E2 -8632.108} C_VEL
LIN {X 0,Y 446.294,Z 251.812,A -85,B 0,C 180,E1 -8632.998,E2 -8632.998} C_VEL
LIN {X 0,Y 446.079,Z 258.376,A -85,B 0,C 180,E1 -8633.895,E2 -8633.895} C_VEL
LIN {X 0,Y 445.921,Z 264.797,A -85,B 0,C 180,E1 -8635.027,E2 -8635.027} C_VEL
LIN {X 0,Y 445.761,Z 270.403,A -85,B 0,C 180,E1 -8636.384,E2 -8636.384} C_VEL
LIN {X 0,Y 445.583,Z 273.105,A -85,B 0,C 180,E1 -8637.288,E2 -8637.288} C_VEL
LIN {X 0,Y 445.489,Z 275.053,A -85,B 0,C 180,E1 -8638.192,E2 -8638.192} C_VEL
LIN {X 0,Y 445.449,Z 276.295,A -85,B 0,C 180,E1 -8639.096,E2 -8639.096} C_VEL
LIN {X 0,Y 445.425,Z 276.862,A -85,B 0,C 180,E1 -8640,E2 -8640} C_VEL
LIN {X 0,Y 445.45,Z 276.755,A -85,B 0,C 180,E1 -8640.904,E2 -8640.904} C_VEL
LIN {X 0,Y 445.54,Z 275.977,A -85,B 0,C 180,E1 -8641.808,E2 -8641.808} C_VEL
LIN {X 0,Y 445.784,Z 273.519,A -85,B 0,C 180,E1 -8643.163,E2 -8643.163} C_VEL
LIN {X 0,Y 445.962,Z 270.97,A -85,B 0,C 180,E1 -8644.067,E2 -8644.067} C_VEL
LIN {X 0,Y 446.128,Z 266.645,A -85,B 0,C 180,E1 -8645.197,E2 -8645.197} C_VEL
LIN {X 0,Y 446.238,Z 260.876,A -85,B 0,C 180,E1 -8646.33,E2 -8646.33} C_VEL
LIN {X 0,Y 446.657,Z 253.894,A -85,B 0,C 180,E1 -8647.371,E2 -8647.371} C_VEL
LIN {X 0,Y 447.078,Z 246.398,A -85,B 0,C 180,E1 -8648.247,E2 -8648.247} C_VEL
LIN {X 0,Y 447.515,Z 237.818,A -85,B 0,C 180,E1 -8649.036,E2 -8649.036} C_VEL
LIN {X 0,Y 447.722,Z 228.312,A -85,B 0,C 180,E1 -8649.715,E2 -8649.715} C_VEL
LIN {X 0,Y 446.221,Z 218.037,A -85,B 0,C 180,E1 -8650.321,E2 -8650.321} C_VEL
LIN {X 0,Y 445.883,Z 215.972,A -85,B 0,C 180,E1 -8650.443,E2 -8650.443} C_VEL
LIN {X 0,Y 446.129,Z 207.649,A -85,B 0,C 180,E1 -8653.668,E2 -8653.668} C_VEL
LIN {X 0,Y 446.461,Z 199.379,A -85,B 0,C 180,E1 -8656.931,E2 -8656.931} C_VEL
LIN {X 0,Y 446.774,Z 191.223,A -85,B 0,C 180,E1 -8660.247,E2 -8660.247} C_VEL
LIN {X 0,Y 447.149,Z 184.314,A -85,B 0,C 180,E1 -8663.137,E2 -8663.137} C_VEL
LIN {X 0,Y 447.723,Z 176.541,A -85,B 0,C 180,E1 -8666.523,E2 -8666.523} C_VEL
LIN {X 0,Y 448.244,Z 170.995,A -85,B 0,C 180,E1 -8669.081,E2 -8669.081} C_VEL
LIN {X 0,Y 448.361,Z 166.8,A -85,B 0,C 180,E1 -8671.15,E2 -8671.15} C_VEL
LIN {X 0,Y 447.619,Z 162.358,A -85,B 0,C 180,E1 -8673.679,E2 -8673.679} C_VEL
LIN {X 0,Y 446.599,Z 157.832,A -85,B 0,C 180,E1 -8676.727,E2 -8676.727} C_VEL
LIN {X 0,Y 446.434,Z 156.878,A -85,B 0,C 180,E1 -8677.591,E2 -8677.591} C_VEL
LIN {X 0,Y 446.45,Z 156.876,A -85,B 0,C 180,E1 -8680.197,E2 -8680.197} C_VEL
LIN {X 0,Y 446.434,Z 156.877,A -85,B 0,C 180,E1 -8682.604,E2 -8682.604} C_VEL
LIN {X 0,Y 446.457,Z 156.875,A -85,B 0,C 180,E1 -8685.103,E2 -8685.103} C_VEL
LIN {X 0,Y 446.434,Z 156.877,A -85,B 0,C 180,E1 -8688.608,E2 -8688.608} C_VEL
LIN {X 0,Y 446.45,Z 156.876,A -85,B 0,C 180,E1 -8690.972,E2 -8690.972} C_VEL
LIN {X 0,Y 446.434,Z 156.94,A -85,B 0,C 180,E1 -8693.257,E2 -8693.257} C_VEL
LIN {X 0,Y 447.335,Z 160.635,A -85,B 0,C 180,E1 -8695.556,E2 -8695.556} C_VEL
LIN {X 0,Y 448.645,Z 166.339,A -85,B 0,C 180,E1 -8698.359,E2 -8698.359} C_VEL
LIN {X 0,Y 450.007,Z 173.027,A -85,B 0,C 180,E1 -8701.042,E2 -8701.042} C_VEL
LIN {X 0,Y 450.377,Z 175.931,A -85,B 0,C 180,E1 -8702.085,E2 -8702.085} C_VEL
LIN {X 0,Y 449.677,Z 182.229,A -85,B 0,C 180,E1 -8704.047,E2 -8704.047} C_VEL
LIN {X 0,Y 448.346,Z 193.843,A -85,B 0,C 180,E1 -8707.382,E2 -8707.382} C_VEL
LIN {X 0,Y 447.39,Z 206.442,A -85,B 0,C 180,E1 -8710.737,E2 -8710.737} C_VEL
LIN {X 0,Y 446.559,Z 220.492,A -85,B 0,C 180,E1 -8714.269,E2 -8714.269} C_VEL
LIN {X 0,Y 448.173,Z 232.514,A -85,B 0,C 180,E1 -8714.669,E2 -8714.669} C_VEL
LIN {X 0,Y 448.679,Z 241.197,A -85,B 0,C 180,E1 -8715.021,E2 -8715.021} C_VEL
LIN {X 0,Y 448.189,Z 254.443,A -85,B 0,C 180,E1 -8715.7,E2 -8715.7} C_VEL
LIN {X 0,Y 447.65,Z 265.854,A -85,B 0,C 180,E1 -8716.477,E2 -8716.477} C_VEL
LIN {X 0,Y 447.106,Z 276.534,A -85,B 0,C 180,E1 -8717.401,E2 -8717.401} C_VEL
LIN {X 0,Y 446.701,Z 286.125,A -85,B 0,C 180,E1 -8718.427,E2 -8718.427} C_VEL
LIN {X 0,Y 446.238,Z 294.852,A -85,B 0,C 180,E1 -8719.564,E2 -8719.564} C_VEL
LIN {X 0,Y 445.903,Z 303.278,A -85,B 0,C 180,E1 -8720.93,E2 -8720.93} C_VEL
LIN {X 0,Y 445.672,Z 310.054,A -85,B 0,C 180,E1 -8722.296,E2 -8722.296} C_VEL
LIN {X 0,Y 445.511,Z 315.435,A -85,B 0,C 180,E1 -8723.659,E2 -8723.659} C_VEL
LIN {X 0,Y 445.488,Z 319.595,A -85,B 0,C 180,E1 -8725.021,E2 -8725.021} C_VEL
LIN {X 0,Y 445.424,Z 322.651,A -85,B 0,C 180,E1 -8726.38,E2 -8726.38} C_VEL
LIN {X 0,Y 445.468,Z 324.11,A -85,B 0,C 180,E1 -8727.286,E2 -8727.286} C_VEL
LIN {X 0,Y 445.426,Z 325.142,A -85,B 0,C 180,E1 -8728.19,E2 -8728.19} C_VEL
LIN {X 0,Y 445.431,Z 325.775,A -85,B 0,C 180,E1 -8729.095,E2 -8729.095} C_VEL
LIN {X 0,Y 445.41,Z 325.965,A -85,B 0,C 180,E1 -8729.999,E2 -8729.999} C_VEL
LIN {X 0,Y 445.432,Z 325.724,A -85,B 0,C 180,E1 -8730.903,E2 -8730.903} C_VEL
LIN {X 0,Y 445.45,Z 325.081,A -85,B 0,C 180,E1 -8731.807,E2 -8731.807} C_VEL
LIN {X 0,Y 445.468,Z 324.02,A -85,B 0,C 180,E1 -8732.711,E2 -8732.711} C_VEL
LIN {X 0,Y 445.44,Z 322.479,A -85,B 0,C 180,E1 -8733.617,E2 -8733.617} C_VEL
LIN {X 0,Y 445.484,Z 319.337,A -85,B 0,C 180,E1 -8734.976,E2 -8734.976} C_VEL
LIN {X 0,Y 445.528,Z 314.909,A -85,B 0,C 180,E1 -8736.384,E2 -8736.384} C_VEL
LIN {X 0,Y 445.697,Z 308.545,A -85,B 0,C 180,E1 -8737.929,E2 -8737.929} C_VEL
LIN {X 0,Y 445.935,Z 301.29,A -85,B 0,C 180,E1 -8739.295,E2 -8739.295} C_VEL
LIN {X 0,Y 446.3,Z 292.23,A -85,B 0,C 180,E1 -8740.661,E2 -8740.661} C_VEL
LIN {X 0,Y 446.697,Z 282.772,A -85,B 0,C 180,E1 -8741.801,E2 -8741.801} C_VEL
LIN {X 0,Y 447.222,Z 271.939,A -85,B 0,C 180,E1 -8742.85,E2 -8742.85} C_VEL
LIN {X 0,Y 447.653,Z 262.058,A -85,B 0,C 180,E1 -8743.619,E2 -8743.619} C_VEL
LIN {X 0,Y 448.085,Z 249.92,A -85,B 0,C 180,E1 -8744.358,E2 -8744.358} C_VEL
LIN {X 0,Y 448.354,Z 237.579,A -85,B 0,C 180,E1 -8744.915,E2 -8744.915} C_VEL
LIN {X 0,Y 446.934,Z 224.807,A -85,B 0,C 180,E1 -8745.346,E2 -8745.346} C_VEL
LIN {X 0,Y 446.417,Z 220.473,A -85,B 0,C 180,E1 -8745.463,E2 -8745.463} C_VEL
LIN {X 0,Y 447.075,Z 206.697,A -85,B 0,C 180,E1 -8748.798,E2 -8748.798} C_VEL
LIN {X 0,Y 447.836,Z 192.891,A -85,B 0,C 180,E1 -8752.195,E2 -8752.195} C_VEL
LIN {X 0,Y 448.762,Z 179.701,A -85,B 0,C 180,E1 -8755.508,E2 -8755.508} C_VEL
LIN {X 0,Y 449.229,Z 172.011,A -85,B 0,C 180,E1 -8757.483,E2 -8757.483} C_VEL
LIN {X 0,Y 448.293,Z 166.198,A -85,B 0,C 180,E1 -8759.076,E2 -8759.076} C_VEL
LIN {X 0,Y 446.418,Z 156.879,A -85,B 0,C 180,E1 -8761.774,E2 -8761.774} C_VEL
LIN {X 0,Y 446.425,Z 156.879,A -85,B 0,C 180,E1 -8764.521,E2 -8764.521} C_VEL
LIN {X 0,Y 446.42,Z 156.877,A -85,B 0,C 180,E1 -8768.08,E2 -8768.08} C_VEL
LIN {X 0,Y 446.409,Z 156.876,A -85,B 0,C 180,E1 -8771.391,E2 -8771.391} C_VEL
LIN {X 0,Y 446.447,Z 156.873,A -85,B 0,C 180,E1 -8775.102,E2 -8775.102} C_VEL
LIN {X 0,Y 446.434,Z 156.876,A -85,B 0,C 180,E1 -8778.609,E2 -8778.609} C_VEL
LIN {X 0,Y 446.463,Z 156.872,A -85,B 0,C 180,E1 -8780.975,E2 -8780.975} C_VEL
LIN {X 0,Y 446.405,Z 156.88,A -85,B 0,C 180,E1 -8784.372,E2 -8784.372} C_VEL
LIN {X 0,Y 446.411,Z 156.88,A -85,B 0,C 180,E1 -8787.637,E2 -8787.637} C_VEL
LIN {X 0,Y 446.457,Z 156.873,A -85,B 0,C 180,E1 -8790.791,E2 -8790.791} C_VEL
LIN {X 0,Y 446.464,Z 156.872,A -85,B 0,C 180,E1 -8793.847,E2 -8793.847} C_VEL
LIN {X 0,Y 446.414,Z 156.875,A -85,B 0,C 180,E1 -8796.822,E2 -8796.822} C_VEL
LIN {X 0,Y 446.43,Z 156.877,A -85,B 0,C 180,E1 -8799.736,E2 -8799.736} C_VEL
LIN {X 0,Y 446.45,Z 156.874,A -85,B 0,C 180,E1 -8802.596,E2 -8802.596} C_VEL
LIN {X 0,Y 446.456,Z 156.873,A -85,B 0,C 180,E1 -8805.412,E2 -8805.412} C_VEL
LIN {X 0,Y 446.523,Z 156.863,A -85,B 0,C 180,E1 -8808.193,E2 -8808.193} C_VEL
LIN {X 0,Y 446.584,Z 156.855,A -85,B 0,C 180,E1 -8811.857,E2 -8811.857} C_VEL
LIN {X 0,Y 446.635,Z 156.852,A -85,B 0,C 180,E1 -8814.582,E2 -8814.582} C_VEL
LIN {X 0,Y 446.697,Z 156.844,A -85,B 0,C 180,E1 -8817.295,E2 -8817.295} C_VEL
LIN {X 0,Y 446.777,Z 156.832,A -85,B 0,C 180,E1 -8820,E2 -8820} C_VEL
LIN {X 0,Y 446.671,Z 156.847,A -85,B 0,C 180,E1 -8822.705,E2 -8822.705} C_VEL
LIN {X 0,Y 446.631,Z 156.853,A -85,B 0,C 180,E1 -8826.324,E2 -8826.324} C_VEL
LIN {X 0,Y 446.525,Z 156.865,A -85,B 0,C 180,E1 -8829.056,E2 -8829.056} C_VEL
LIN {X 0,Y 446.519,Z 156.868,A -85,B 0,C 180,E1 -8832.73,E2 -8832.73} C_VEL
LIN {X 0,Y 446.475,Z 156.872,A -85,B 0,C 180,E1 -8836.46,E2 -8836.46} C_VEL
LIN {X 0,Y 446.456,Z 156.873,A -85,B 0,C 180,E1 -8839.304,E2 -8839.304} C_VEL
LIN {X 0,Y 446.423,Z 156.877,A -85,B 0,C 180,E1 -8842.199,E2 -8842.199} C_VEL
LIN {X 0,Y 446.432,Z 156.875,A -85,B 0,C 180,E1 -8845.154,E2 -8845.154} C_VEL
LIN {X 0,Y 446.435,Z 156.877,A -85,B 0,C 180,E1 -8848.182,E2 -8848.182} C_VEL
LIN {X 0,Y 446.404,Z 156.88,A -85,B 0,C 180,E1 -8851.301,E2 -8851.301} C_VEL
LIN {X 0,Y 446.419,Z 156.878,A -85,B 0,C 180,E1 -8854.524,E2 -8854.524} C_VEL
LIN {X 0,Y 446.419,Z 156.879,A -85,B 0,C 180,E1 -8858.083,E2 -8858.083} C_VEL
LIN {X 0,Y 446.416,Z 156.875,A -85,B 0,C 180,E1 -8860.919,E2 -8860.919} C_VEL
LIN {X 0,Y 446.412,Z 156.878,A -85,B 0,C 180,E1 -8863.845,E2 -8863.845} C_VEL
LIN {X 0,Y 446.411,Z 156.878,A -85,B 0,C 180,E1 -8866.402,E2 -8866.402} C_VEL
LIN {X 0,Y 446.433,Z 156.877,A -85,B 0,C 180,E1 -8869.803,E2 -8869.803} C_VEL
LIN {X 0,Y 446.393,Z 156.883,A -85,B 0,C 180,E1 -8873.256,E2 -8873.256} C_VEL
LIN {X 0,Y 446.441,Z 156.875,A -85,B 0,C 180,E1 -8876.568,E2 -8876.568} C_VEL
LIN {X 0,Y 446.436,Z 156.875,A -85,B 0,C 180,E1 -8879.978,E2 -8879.978} C_VEL
LIN {X 0,Y 446.459,Z 156.873,A -85,B 0,C 180,E1 -8882.84,E2 -8882.84} C_VEL
LIN {X 0,Y 446.456,Z 156.87,A -85,B 0,C 180,E1 -8885.927,E2 -8885.927} C_VEL
LIN {X 0,Y 446.45,Z 156.874,A -85,B 0,C 180,E1 -8888.775,E2 -8888.775} C_VEL
LIN {X 0,Y 446.455,Z 156.873,A -85,B 0,C 180,E1 -8891.651,E2 -8891.651} C_VEL
LIN {X 0,Y 446.505,Z 156.867,A -85,B 0,C 180,E1 -8894.481,E2 -8894.481} C_VEL
LIN {X 0,Y 446.516,Z 156.866,A -85,B 0,C 180,E1 -8898.195,E2 -8898.195} C_VEL
LIN {X 0,Y 446.6,Z 156.857,A -85,B 0,C 180,E1 -8901.859,E2 -8901.859} C_VEL
LIN {X 0,Y 446.646,Z 156.85,A -85,B 0,C 180,E1 -8904.584,E2 -8904.584} C_VEL
LIN {X 0,Y 446.617,Z 156.852,A -85,B 0,C 180,E1 -8907.025,E2 -8907.025} C_VEL
LIN {X 0,Y 446.397,Z 156.88,A -85,B 0,C 180,E1 -8907.528,E2 -8907.528} C_VEL
LIN {X 0,Y 445.081,Z 157.047,A -85,B 0,C 180,E1 -8908.271,E2 -8908.271} C_VEL
LIN {X 0,Y 440.628,Z 157.601,A -85,B 0,C 180,E1 -8909.984,E2 -8909.984} C_VEL
LIN {X 0,Y 439.572,Z 157.728,A -85,B 0,C 180,E1 -8910.747,E2 -8910.747} C_VEL
LIN {X 0,Y 439.508,Z 157.735,A -85,B 0,C 180,E1 -8911.006,E2 -8911.006} C_VEL
LIN {X 0,Y 439.634,Z 157.721,A -85,B 0,C 180,E1 -8912.75,E2 -8912.75} C_VEL
LIN {X 0,Y 439.621,Z 157.725,A -85,B 0,C 180,E1 -8916.427,E2 -8916.427} C_VEL
LIN {X 0,Y 439.502,Z 157.739,A -85,B 0,C 180,E1 -8919.203,E2 -8919.203} C_VEL
LIN {X 0,Y 439.468,Z 157.741,A -85,B 0,C 180,E1 -8922.939,E2 -8922.939} C_VEL
LIN {X 0,Y 439.451,Z 157.744,A -85,B 0,C 180,E1 -8926.349,E2 -8926.349} C_VEL
LIN {X 0,Y 439.407,Z 157.751,A -85,B 0,C 180,E1 -8929.627,E2 -8929.627} C_VEL
LIN {X 0,Y 439.367,Z 157.755,A -85,B 0,C 180,E1 -8932.577,E2 -8932.577} C_VEL
LIN {X 0,Y 439.37,Z 157.755,A -85,B 0,C 180,E1 -8935.588,E2 -8935.588} C_VEL
LIN {X 0,Y 439.394,Z 157.754,A -85,B 0,C 180,E1 -8938.676,E2 -8938.676} C_VEL
LIN {X 0,Y 439.373,Z 157.755,A -85,B 0,C 180,E1 -8942.031,E2 -8942.031} C_VEL
LIN {X 0,Y 439.394,Z 157.753,A -85,B 0,C 180,E1 -8945.34,E2 -8945.34} C_VEL
LIN {X 0,Y 439.358,Z 157.759,A -85,B 0,C 180,E1 -8948.599,E2 -8948.599} C_VEL
LIN {X 0,Y 439.363,Z 157.758,A -85,B 0,C 180,E1 -8952.209,E2 -8952.209} C_VEL
LIN {X 0,Y 439.404,Z 157.751,A -85,B 0,C 180,E1 -8955.271,E2 -8955.271} C_VEL
LIN {X 0,Y 439.394,Z 157.754,A -85,B 0,C 180,E1 -8958.744,E2 -8958.744} C_VEL
LIN {X 0,Y 439.363,Z 157.754,A -85,B 0,C 180,E1 -8961.611,E2 -8961.611} C_VEL
LIN {X 0,Y 439.399,Z 157.751,A -85,B 0,C 180,E1 -8964.844,E2 -8964.844} C_VEL
LIN {X 0,Y 439.506,Z 157.902,A -85,B 0,C 180,E1 -8967.533,E2 -8967.533} C_VEL
LIN {X 0,Y 440.207,Z 162.644,A -85,B 0,C 180,E1 -8969.557,E2 -8969.557} C_VEL
LIN {X 0,Y 440.061,Z 168.401,A -85,B 0,C 180,E1 -8971.923,E2 -8971.923} C_VEL
LIN {X 0,Y 439.738,Z 175.917,A -85,B 0,C 180,E1 -8974.942,E2 -8974.942} C_VEL
LIN {X 0,Y 439.39,Z 184.661,A -85,B 0,C 180,E1 -8978.415,E2 -8978.415} C_VEL
LIN {X 0,Y 439.167,Z 192.141,A -85,B 0,C 180,E1 -8981.333,E2 -8981.333} C_VEL
LIN {X 0,Y 438.93,Z 200.844,A -85,B 0,C 180,E1 -8984.681,E2 -8984.681} C_VEL
LIN {X 0,Y 438.728,Z 209.514,A -85,B 0,C 180,E1 -8987.98,E2 -8987.98} C_VEL
LIN {X 0,Y 438.563,Z 215.244,A -85,B 0,C 180,E1 -8990.139,E2 -8990.139} C_VEL
LIN {X 0,Y 439.794,Z 226.245,A -85,B 0,C 180,E1 -8990.689,E2 -8990.689} C_VEL
LIN {X 0,Y 439.99,Z 231.854,A -85,B 0,C 180,E1 -8991.04,E2 -8991.04} C_VEL
LIN {X 0,Y 439.647,Z 240.778,A -85,B 0,C 180,E1 -8991.728,E2 -8991.728} C_VEL
LIN {X 0,Y 439.313,Z 249.864,A -85,B 0,C 180,E1 -8992.647,E2 -8992.647} C_VEL
LIN {X 0,Y 439.073,Z 256.941,A -85,B 0,C 180,E1 -8993.567,E2 -8993.567} C_VEL
LIN {X 0,Y 438.883,Z 263.792,A -85,B 0,C 180,E1 -8994.717,E2 -8994.717} C_VEL
LIN {X 0,Y 438.75,Z 268.968,A -85,B 0,C 180,E1 -8995.866,E2 -8995.866} C_VEL
LIN {X 0,Y 438.513,Z 273.38,A -85,B 0,C 180,E1 -8997.244,E2 -8997.244} C_VEL
LIN {X 0,Y 438.405,Z 275.371,A -85,B 0,C 180,E1 -8998.163,E2 -8998.163} C_VEL
LIN {X 0,Y 438.387,Z 276.654,A -85,B 0,C 180,E1 -8999.081,E2 -8999.081} C_VEL
LIN {X 0,Y 438.362,Z 277.261,A -85,B 0,C 180,E1 -9000,E2 -9000} C_VEL
LIN {X 0,Y 438.389,Z 277.193,A -85,B 0,C 180,E1 -9000.919,E2 -9000.919} C_VEL
LIN {X 0,Y 438.485,Z 276.455,A -85,B 0,C 180,E1 -9001.837,E2 -9001.837} C_VEL
LIN {X 0,Y 438.741,Z 274.062,A -85,B 0,C 180,E1 -9003.214,E2 -9003.214} C_VEL
LIN {X 0,Y 438.921,Z 271.563,A -85,B 0,C 180,E1 -9004.132,E2 -9004.132} C_VEL
LIN {X 0,Y 439.026,Z 268.282,A -85,B 0,C 180,E1 -9005.051,E2 -9005.051} C_VEL
LIN {X 0,Y 439.22,Z 262.906,A -85,B 0,C 180,E1 -9006.201,E2 -9006.201} C_VEL
LIN {X 0,Y 439.608,Z 255.827,A -85,B 0,C 180,E1 -9007.348,E2 -9007.348} C_VEL
LIN {X 0,Y 440.126,Z 247.5,A -85,B 0,C 180,E1 -9008.378,E2 -9008.378} C_VEL
LIN {X 0,Y 440.579,Z 239.171,A -85,B 0,C 180,E1 -9009.179,E2 -9009.179} C_VEL
LIN {X 0,Y 440.921,Z 230.048,A -85,B 0,C 180,E1 -9009.866,E2 -9009.866} C_VEL
LIN {X 0,Y 439.64,Z 220.475,A -85,B 0,C 180,E1 -9010.477,E2 -9010.477} C_VEL
LIN {X 0,Y 438.887,Z 216.099,A -85,B 0,C 180,E1 -9010.729,E2 -9010.729} C_VEL
LIN {X 0,Y 439.176,Z 206.896,A -85,B 0,C 180,E1 -9014.362,E2 -9014.362} C_VEL
LIN {X 0,Y 439.506,Z 198.661,A -85,B 0,C 180,E1 -9017.687,E2 -9017.687} C_VEL
LIN {X 0,Y 439.914,Z 190.571,A -85,B 0,C 180,E1 -9021.067,E2 -9021.067} C_VEL
LIN {X 0,Y 440.416,Z 182.537,A -85,B 0,C 180,E1 -9024.55,E2 -9024.55} C_VEL
LIN {X 0,Y 441.146,Z 174.917,A -85,B 0,C 180,E1 -9028.033,E2 -9028.033} C_VEL
LIN {X 0,Y 441.552,Z 169.425,A -85,B 0,C 180,E1 -9030.738,E2 -9030.738} C_VEL
LIN {X 0,Y 441.064,Z 165.822,A -85,B 0,C 180,E1 -9032.804,E2 -9032.804} C_VEL
LIN {X 0,Y 440.239,Z 161.692,A -85,B 0,C 180,E1 -9035.493,E2 -9035.493} C_VEL
LIN {X 0,Y 439.439,Z 158.061,A -85,B 0,C 180,E1 -9038.401,E2 -9038.401} C_VEL
LIN {X 0,Y 439.415,Z 157.752,A -85,B 0,C 180,E1 -9039.181,E2 -9039.181} C_VEL
LIN {X 0,Y 439.387,Z 157.755,A -85,B 0,C 180,E1 -9042.626,E2 -9042.626} C_VEL
LIN {X 0,Y 439.406,Z 157.754,A -85,B 0,C 180,E1 -9045.27,E2 -9045.27} C_VEL
LIN {X 0,Y 439.395,Z 157.754,A -85,B 0,C 180,E1 -9048.743,E2 -9048.743} C_VEL
LIN {X 0,Y 439.38,Z 157.757,A -85,B 0,C 180,E1 -9051.607,E2 -9051.607} C_VEL
LIN {X 0,Y 439.397,Z 157.888,A -85,B 0,C 180,E1 -9051.989,E2 -9051.989} C_VEL
LIN {X 0,Y 440.44,Z 162.016,A -85,B 0,C 180,E1 -9054.938,E2 -9054.938} C_VEL
LIN {X 0,Y 441.524,Z 166.863,A -85,B 0,C 180,E1 -9057.526,E2 -9057.526} C_VEL
LIN {X 0,Y 442.721,Z 172.517,A -85,B 0,C 180,E1 -9059.996,E2 -9059.996} C_VEL
LIN {X 0,Y 443.454,Z 176.678,A -85,B 0,C 180,E1 -9061.61,E2 -9061.61} C_VEL
LIN {X 0,Y 443.402,Z 179.662,A -85,B 0,C 180,E1 -9062.634,E2 -9062.634} C_VEL
LIN {X 0,Y 442.093,Z 189.29,A -85,B 0,C 180,E1 -9065.585,E2 -9065.585} C_VEL
LIN {X 0,Y 440.887,Z 201.298,A -85,B 0,C 180,E1 -9068.981,E2 -9068.981} C_VEL
LIN {X 0,Y 440.062,Z 212.112,A -85,B 0,C 180,E1 -9071.854,E2 -9071.854} C_VEL
LIN {X 0,Y 439.597,Z 220.539,A -85,B 0,C 180,E1 -9074.006,E2 -9074.006} C_VEL
LIN {X 0,Y 441.297,Z 232.487,A -85,B 0,C 180,E1 -9074.409,E2 -9074.409} C_VEL
LIN {X 0,Y 441.829,Z 241.354,A -85,B 0,C 180,E1 -9074.783,E2 -9074.783} C_VEL
LIN {X 0,Y 441.3,Z 254.443,A -85,B 0,C 180,E1 -9075.472,E2 -9075.472} C_VEL
LIN {X 0,Y 440.716,Z 265.889,A -85,B 0,C 180,E1 -9076.27,E2 -9076.27} C_VEL
LIN {X 0,Y 440.078,Z 277.553,A -85,B 0,C 180,E1 -9077.314,E2 -9077.314} C_VEL
LIN {X 0,Y 439.635,Z 287.803,A -85,B 0,C 180,E1 -9078.472,E2 -9078.472} C_VEL
LIN {X 0,Y 439.039,Z 297.615,A -85,B 0,C 180,E1 -9079.857,E2 -9079.857} C_VEL
LIN {X 0,Y 438.758,Z 305.437,A -85,B 0,C 180,E1 -9081.246,E2 -9081.246} C_VEL
LIN {X 0,Y 438.524,Z 311.676,A -85,B 0,C 180,E1 -9082.632,E2 -9082.632} C_VEL
LIN {X 0,Y 438.374,Z 316.519,A -85,B 0,C 180,E1 -9083.991,E2 -9083.991} C_VEL
LIN {X 0,Y 438.356,Z 320.364,A -85,B 0,C 180,E1 -9085.401,E2 -9085.401} C_VEL
LIN {X 0,Y 438.325,Z 322.298,A -85,B 0,C 180,E1 -9086.321,E2 -9086.321} C_VEL
LIN {X 0,Y 438.392,Z 323.744,A -85,B 0,C 180,E1 -9087.242,E2 -9087.242} C_VEL
LIN {X 0,Y 438.344,Z 324.768,A -85,B 0,C 180,E1 -9088.161,E2 -9088.161} C_VEL
LIN {X 0,Y 438.34,Z 325.39,A -85,B 0,C 180,E1 -9089.08,E2 -9089.08} C_VEL
LIN {X 0,Y 438.348,Z 325.558,A -85,B 0,C 180,E1 -9089.999,E2 -9089.999} C_VEL
LIN {X 0,Y 438.37,Z 325.305,A -85,B 0,C 180,E1 -9090.917,E2 -9090.917} C_VEL
LIN {X 0,Y 438.366,Z 324.649,A -85,B 0,C 180,E1 -9091.836,E2 -9091.836} C_VEL
LIN {X 0,Y 438.394,Z 323.56,A -85,B 0,C 180,E1 -9092.755,E2 -9092.755} C_VEL
LIN {X 0,Y 438.343,Z 321.999,A -85,B 0,C 180,E1 -9093.676,E2 -9093.676} C_VEL
LIN {X 0,Y 438.414,Z 318.821,A -85,B 0,C 180,E1 -9095.057,E2 -9095.057} C_VEL
LIN {X 0,Y 438.447,Z 314.512,A -85,B 0,C 180,E1 -9096.441,E2 -9096.441} C_VEL
LIN {X 0,Y 438.588,Z 308.957,A -85,B 0,C 180,E1 -9097.827,E2 -9097.827} C_VEL
LIN {X 0,Y 438.818,Z 301.938,A -85,B 0,C 180,E1 -9099.214,E2 -9099.214} C_VEL
LIN {X 0,Y 439.167,Z 293.068,A -85,B 0,C 180,E1 -9100.603,E2 -9100.603} C_VEL
LIN {X 0,Y 439.639,Z 283.939,A -85,B 0,C 180,E1 -9101.759,E2 -9101.759} C_VEL
LIN {X 0,Y 440.109,Z 273.719,A -85,B 0,C 180,E1 -9102.799,E2 -9102.799} C_VEL
LIN {X 0,Y 440.49,Z 263.799,A -85,B 0,C 180,E1 -9103.618,E2 -9103.618} C_VEL
LIN {X 0,Y 441.023,Z 251.5,A -85,B 0,C 180,E1 -9104.416,E2 -9104.416} C_VEL
LIN {X 0,Y 441.407,Z 238.728,A -85,B 0,C 180,E1 -9105.022,E2 -9105.022} C_VEL
LIN {X 0,Y 439.967,Z 225.644,A -85,B 0,C 180,E1 -9105.488,E2 -9105.488} C_VEL
LIN {X 0,Y 439.363,Z 220.471,A -85,B 0,C 180,E1 -9105.629,E2 -9105.629} C_VEL
LIN {X 0,Y 440.077,Z 206.361,A -85,B 0,C 180,E1 -9109.108,E2 -9109.108} C_VEL
LIN {X 0,Y 441.037,Z 190.994,A -85,B 0,C 180,E1 -9112.978,E2 -9112.978} C_VEL
LIN {X 0,Y 442.036,Z 177.542,A -85,B 0,C 180,E1 -9116.433,E2 -9116.433} C_VEL
LIN {X 0,Y 442.265,Z 173.704,A -85,B 0,C 180,E1 -9117.439,E2 -9117.439} C_VEL
LIN {X 0,Y 441.512,Z 168.443,A -85,B 0,C 180,E1 -9118.896,E2 -9118.896} C_VEL
LIN {X 0,Y 439.367,Z 157.758,A -85,B 0,C 180,E1 -9122.029,E2 -9122.029} C_VEL
LIN {X 0,Y 439.39,Z 157.756,A -85,B 0,C 180,E1 -9125.339,E2 -9125.339} C_VEL
LIN {X 0,Y 439.367,Z 157.756,A -85,B 0,C 180,E1 -9128.594,E2 -9128.594} C_VEL
LIN {X 0,Y 439.372,Z 157.753,A -85,B 0,C 180,E1 -9131.254,E2 -9131.254} C_VEL
LIN {X 0,Y 439.392,Z 157.752,A -85,B 0,C 180,E1 -9134.728,E2 -9134.728} C_VEL
LIN {X 0,Y 439.403,Z 157.752,A -85,B 0,C 180,E1 -9137.796,E2 -9137.796} C_VEL
LIN {X 0,Y 439.441,Z 157.747,A -85,B 0,C 180,E1 -9140.229,E2 -9140.229} C_VEL
LIN {X 0,Y 439.36,Z 157.755,A -85,B 0,C 180,E1 -9143.711,E2 -9143.711} C_VEL
LIN {X 0,Y 439.361,Z 157.755,A -85,B 0,C 180,E1 -9147.053,E2 -9147.053} C_VEL
LIN {X 0,Y 439.384,Z 157.754,A -85,B 0,C 180,E1 -9150.274,E2 -9150.274} C_VEL
LIN {X 0,Y 439.42,Z 157.749,A -85,B 0,C 180,E1 -9153.588,E2 -9153.588} C_VEL
LIN {X 0,Y 439.371,Z 157.753,A -85,B 0,C 180,E1 -9156.429,E2 -9156.429} C_VEL
LIN {X 0,Y 439.374,Z 157.757,A -85,B 0,C 180,E1 -9159.396,E2 -9159.396} C_VEL
LIN {X 0,Y 439.418,Z 157.75,A -85,B 0,C 180,E1 -9162.309,E2 -9162.309} C_VEL
LIN {X 0,Y 439.433,Z 157.747,A -85,B 0,C 180,E1 -9165.173,E2 -9165.173} C_VEL
LIN {X 0,Y 439.491,Z 157.74,A -85,B 0,C 180,E1 -9168.001,E2 -9168.001} C_VEL
LIN {X 0,Y 439.532,Z 157.734,A -85,B 0,C 180,E1 -9171.726,E2 -9171.726} C_VEL
LIN {X 0,Y 439.61,Z 157.726,A -85,B 0,C 180,E1 -9174.496,E2 -9174.496} C_VEL
LIN {X 0,Y 439.621,Z 157.724,A -85,B 0,C 180,E1 -9178.168,E2 -9178.168} C_VEL
LIN {X 0,Y 439.747,Z 157.707,A -85,B 0,C 180,E1 -9180,E2 -9180} C_VEL
LIN {X 0,Y 439.621,Z 157.726,A -85,B 0,C 180,E1 -9182.749,E2 -9182.749} C_VEL
LIN {X 0,Y 439.603,Z 157.729,A -85,B 0,C 180,E1 -9186.425,E2 -9186.425} C_VEL
LIN {X 0,Y 439.487,Z 157.743,A -85,B 0,C 180,E1 -9189.202,E2 -9189.202} C_VEL
LIN {X 0,Y 439.489,Z 157.743,A -85,B 0,C 180,E1 -9192.727,E2 -9192.727} C_VEL
LIN {X 0,Y 439.433,Z 157.751,A -85,B 0,C 180,E1 -9196.349,E2 -9196.349} C_VEL
LIN {X 0,Y 439.42,Z 157.749,A -85,B 0,C 180,E1 -9199.625,E2 -9199.625} C_VEL
LIN {X 0,Y 439.363,Z 157.758,A -85,B 0,C 180,E1 -9202.576,E2 -9202.576} C_VEL
LIN {X 0,Y 439.368,Z 157.754,A -85,B 0,C 180,E1 -9205.587,E2 -9205.587} C_VEL
LIN {X 0,Y 439.386,Z 157.751,A -85,B 0,C 180,E1 -9208.676,E2 -9208.676} C_VEL
LIN {X 0,Y 439.358,Z 157.757,A -85,B 0,C 180,E1 -9212.032,E2 -9212.032} C_VEL
LIN {X 0,Y 439.384,Z 157.754,A -85,B 0,C 180,E1 -9215.342,E2 -9215.342} C_VEL
LIN {X 0,Y 439.378,Z 157.753,A -85,B 0,C 180,E1 -9218.595,E2 -9218.595} C_VEL
LIN {X 0,Y 439.377,Z 157.755,A -85,B 0,C 180,E1 -9221.258,E2 -9221.258} C_VEL
LIN {X 0,Y 439.396,Z 157.752,A -85,B 0,C 180,E1 -9224.73,E2 -9224.73} C_VEL
LIN {X 0,Y 439.389,Z 157.755,A -85,B 0,C 180,E1 -9227.797,E2 -9227.797} C_VEL
LIN {X 0,Y 439.386,Z 157.752,A -85,B 0,C 180,E1 -9230.225,E2 -9230.225} C_VEL
LIN {X 0,Y 439.365,Z 157.755,A -85,B 0,C 180,E1 -9233.714,E2 -9233.714} C_VEL
LIN {X 0,Y 439.366,Z 157.757,A -85,B 0,C 180,E1 -9237.056,E2 -9237.056} C_VEL
LIN {X 0,Y 439.391,Z 157.753,A -85,B 0,C 180,E1 -9240.277,E2 -9240.277} C_VEL
LIN {X 0,Y 439.414,Z 157.75,A -85,B 0,C 180,E1 -9243.397,E2 -9243.397} C_VEL
LIN {X 0,Y 439.378,Z 157.755,A -85,B 0,C 180,E1 -9246.431,E2 -9246.431} C_VEL
LIN {X 0,Y 439.385,Z 157.753,A -85,B 0,C 180,E1 -9249.399,E2 -9249.399} C_VEL
LIN {X 0,Y 439.43,Z 157.748,A -85,B 0,C 180,E1 -9252.311,E2 -9252.311} C_VEL
LIN {X 0,Y 439.443,Z 157.746,A -85,B 0,C 180,E1 -9255.176,E2 -9255.176} C_VEL
LIN {X 0,Y 439.482,Z 157.741,A -85,B 0,C 180,E1 -9258.003,E2 -9258.003} C_VEL
LIN {X 0,Y 439.548,Z 157.734,A -85,B 0,C 180,E1 -9261.728,E2 -9261.728} C_VEL
LIN {X 0,Y 439.622,Z 157.725,A -85,B 0,C 180,E1 -9264.497,E2 -9264.497} C_VEL
LIN {X 0,Y 439.635,Z 157.724,A -85,B 0,C 180,E1 -9268.169,E2 -9268.169} C_VEL
LIN {X 0,Y 439.689,Z 157.718,A -85,B 0,C 180,E1 -9270.001,E2 -9270.001} C_VEL
LIN {X 0,Y 439.508,Z 157.735,A -85,B 0,C 180,E1 -9271.006,E2 -9271.006} C_VEL
LIN {X 0,Y 438.869,Z 157.82,A -85,B 0,C 180,E1 -9271.771,E2 -9271.771} C_VEL
LIN {X 0,Y 435.936,Z 158.182,A -85,B 0,C 180,E1 -9273.012,E2 -9273.012} C_VEL
LIN {X 0,Y 433.481,Z 158.489,A -85,B 0,C 180,E1 -9274.014,E2 -9274.014} C_VEL
LIN {X 0,Y 432.504,Z 158.61,A -85,B 0,C 180,E1 -9274.789,E2 -9274.789} C_VEL
LIN {X 0,Y 432.468,Z 158.614,A -85,B 0,C 180,E1 -9275.051,E2 -9275.051} C_VEL
LIN {X 0,Y 432.589,Z 158.6,A -85,B 0,C 180,E1 -9277.68,E2 -9277.68} C_VEL
LIN {X 0,Y 432.394,Z 158.624,A -85,B 0,C 180,E1 -9281.249,E2 -9281.249} C_VEL
LIN {X 0,Y 432.371,Z 158.625,A -85,B 0,C 180,E1 -9284.113,E2 -9284.113} C_VEL
LIN {X 0,Y 432.399,Z 158.625,A -85,B 0,C 180,E1 -9287.013,E2 -9287.013} C_VEL
LIN {X 0,Y 432.343,Z 158.632,A -85,B 0,C 180,E1 -9289.962,E2 -9289.962} C_VEL
LIN {X 0,Y 432.316,Z 158.634,A -85,B 0,C 180,E1 -9292.966,E2 -9292.966} C_VEL
LIN {X 0,Y 432.321,Z 158.63,A -85,B 0,C 180,E1 -9296.036,E2 -9296.036} C_VEL
LIN {X 0,Y 432.331,Z 158.632,A -85,B 0,C 180,E1 -9299.19,E2 -9299.19} C_VEL
LIN {X 0,Y 432.327,Z 158.634,A -85,B 0,C 180,E1 -9302.444,E2 -9302.444} C_VEL
LIN {X 0,Y 432.346,Z 158.63,A -85,B 0,C 180,E1 -9305.632,E2 -9305.632} C_VEL
LIN {X 0,Y 432.323,Z 158.636,A -85,B 0,C 180,E1 -9308.711,E2 -9308.711} C_VEL
LIN {X 0,Y 432.314,Z 158.633,A -85,B 0,C 180,E1 -9311.801,E2 -9311.801} C_VEL
LIN {X 0,Y 432.339,Z 158.632,A -85,B 0,C 180,E1 -9314.348,E2 -9314.348} C_VEL
LIN {X 0,Y 432.325,Z 158.634,A -85,B 0,C 180,E1 -9317.016,E2 -9317.016} C_VEL
LIN {X 0,Y 432.32,Z 158.632,A -85,B 0,C 180,E1 -9319.824,E2 -9319.824} C_VEL
LIN {X 0,Y 432.303,Z 158.634,A -85,B 0,C 180,E1 -9323.022,E2 -9323.022} C_VEL
LIN {X 0,Y 432.363,Z 158.629,A -85,B 0,C 180,E1 -9325.997,E2 -9325.997} C_VEL
LIN {X 0,Y 432.457,Z 158.833,A -85,B 0,C 180,E1 -9327.43,E2 -9327.43} C_VEL
LIN {X 0,Y 433.193,Z 164.336,A -85,B 0,C 180,E1 -9329.806,E2 -9329.806} C_VEL
LIN {X 0,Y 432.947,Z 171.987,A -85,B 0,C 180,E1 -9332.966,E2 -9332.966} C_VEL
LIN {X 0,Y 432.52,Z 180.812,A -85,B 0,C 180,E1 -9336.541,E2 -9336.541} C_VEL
LIN {X 0,Y 432.241,Z 189.598,A -85,B 0,C 180,E1 -9340.035,E2 -9340.035} C_VEL
LIN {X 0,Y 431.925,Z 199.048,A -85,B 0,C 180,E1 -9343.744,E2 -9343.744} C_VEL
LIN {X 0,Y 431.675,Z 208.266,A -85,B 0,C 180,E1 -9347.304,E2 -9347.304} C_VEL
LIN {X 0,Y 431.496,Z 215.455,A -85,B 0,C 180,E1 -9350.005,E2 -9350.005} C_VEL
LIN {X 0,Y 432.687,Z 226.003,A -85,B 0,C 180,E1 -9350.534,E2 -9350.534} C_VEL
LIN {X 0,Y 432.986,Z 231.675,A -85,B 0,C 180,E1 -9350.894,E2 -9350.894} C_VEL
LIN {X 0,Y 432.609,Z 240.681,A -85,B 0,C 180,E1 -9351.593,E2 -9351.593} C_VEL
LIN {X 0,Y 432.27,Z 249.848,A -85,B 0,C 180,E1 -9352.527,E2 -9352.527} C_VEL
LIN {X 0,Y 432.027,Z 257.001,A -85,B 0,C 180,E1 -9353.461,E2 -9353.461} C_VEL
LIN {X 0,Y 431.812,Z 263.928,A -85,B 0,C 180,E1 -9354.63,E2 -9354.63} C_VEL
LIN {X 0,Y 431.686,Z 269.168,A -85,B 0,C 180,E1 -9355.799,E2 -9355.799} C_VEL
LIN {X 0,Y 431.445,Z 273.645,A -85,B 0,C 180,E1 -9357.199,E2 -9357.199} C_VEL
LIN {X 0,Y 431.325,Z 275.679,A -85,B 0,C 180,E1 -9358.133,E2 -9358.133} C_VEL
LIN {X 0,Y 431.297,Z 277.008,A -85,B 0,C 180,E1 -9359.066,E2 -9359.066} C_VEL
LIN {X 0,Y 431.301,Z 277.658,A -85,B 0,C 180,E1 -9360,E2 -9360} C_VEL
LIN {X 0,Y 431.33,Z 277.637,A -85,B 0,C 180,E1 -9360.934,E2 -9360.934} C_VEL
LIN {X 0,Y 431.433,Z 276.942,A -85,B 0,C 180,E1 -9361.867,E2 -9361.867} C_VEL
LIN {X 0,Y 431.7,Z 274.621,A -85,B 0,C 180,E1 -9363.267,E2 -9363.267} C_VEL
LIN {X 0,Y 431.882,Z 272.179,A -85,B 0,C 180,E1 -9364.2,E2 -9364.2} C_VEL
LIN {X 0,Y 431.995,Z 268.961,A -85,B 0,C 180,E1 -9365.134,E2 -9365.134} C_VEL
LIN {X 0,Y 432.205,Z 263.689,A -85,B 0,C 180,E1 -9366.302,E2 -9366.302} C_VEL
LIN {X 0,Y 432.639,Z 256.742,A -85,B 0,C 180,E1 -9367.467,E2 -9367.467} C_VEL
LIN {X 0,Y 433.176,Z 248.62,A -85,B 0,C 180,E1 -9368.514,E2 -9368.514} C_VEL
LIN {X 0,Y 433.76,Z 239.251,A -85,B 0,C 180,E1 -9369.442,E2 -9369.442} C_VEL
LIN {X 0,Y 434.104,Z 231.787,A -85,B 0,C 180,E1 -9370.023,E2 -9370.023} C_VEL
LIN {X 0,Y 432.846,Z 221.786,A -85,B 0,C 180,E1 -9370.702,E2 -9370.702} C_VEL
LIN {X 0,Y 431.851,Z 216.236,A -85,B 0,C 180,E1 -9371.024,E2 -9371.024} C_VEL
LIN {X 0,Y 432.171,Z 207.358,A -85,B 0,C 180,E1 -9374.6,E2 -9374.6} C_VEL
LIN {X 0,Y 432.527,Z 199.163,A -85,B 0,C 180,E1 -9377.983,E2 -9377.983} C_VEL
LIN {X 0,Y 432.971,Z 191.11,A -85,B 0,C 180,E1 -9381.421,E2 -9381.421} C_VEL
LIN {X 0,Y 433.531,Z 183.243,A -85,B 0,C 180,E1 -9384.929,E2 -9384.929} C_VEL
LIN {X 0,Y 434.346,Z 175.646,A -85,B 0,C 180,E1 -9388.511,E2 -9388.511} C_VEL
LIN {X 0,Y 434.644,Z 172.543,A -85,B 0,C 180,E1 -9390.083,E2 -9390.083} C_VEL
LIN {X 0,Y 434.414,Z 168.676,A -85,B 0,C 180,E1 -9392.268,E2 -9392.268} C_VEL
LIN {X 0,Y 433.732,Z 165.127,A -85,B 0,C 180,E1 -9394.55,E2 -9394.55} C_VEL
LIN {X 0,Y 433.028,Z 161.564,A -85,B 0,C 180,E1 -9397.318,E2 -9397.318} C_VEL
LIN {X 0,Y 432.555,Z 159.496,A -85,B 0,C 180,E1 -9399.321,E2 -9399.321} C_VEL
LIN {X 0,Y 432.33,Z 158.635,A -85,B 0,C 180,E1 -9400.56,E2 -9400.56} C_VEL
LIN {X 0,Y 432.323,Z 158.635,A -85,B 0,C 180,E1 -9403.061,E2 -9403.061} C_VEL
LIN {X 0,Y 432.339,Z 158.632,A -85,B 0,C 180,E1 -9405.664,E2 -9405.664} C_VEL
LIN {X 0,Y 432.339,Z 158.633,A -85,B 0,C 180,E1 -9408.397,E2 -9408.397} C_VEL
LIN {X 0,Y 432.399,Z 158.821,A -85,B 0,C 180,E1 -9410.36,E2 -9410.36} C_VEL
LIN {X 0,Y 433.115,Z 161.804,A -85,B 0,C 180,E1 -9413.101,E2 -9413.101} C_VEL
LIN {X 0,Y 434.054,Z 165.737,A -85,B 0,C 180,E1 -9415.667,E2 -9415.667} C_VEL
LIN {X 0,Y 434.936,Z 169.757,A -85,B 0,C 180,E1 -9417.774,E2 -9417.774} C_VEL
LIN {X 0,Y 435.992,Z 174.763,A -85,B 0,C 180,E1 -9420.018,E2 -9420.018} C_VEL
LIN {X 0,Y 436.66,Z 178.901,A -85,B 0,C 180,E1 -9421.652,E2 -9421.652} C_VEL
LIN {X 0,Y 436.483,Z 182.014,A -85,B 0,C 180,E1 -9422.734,E2 -9422.734} C_VEL
LIN {X 0,Y 435.109,Z 191.438,A -85,B 0,C 180,E1 -9425.676,E2 -9425.676} C_VEL
LIN {X 0,Y 433.844,Z 203.361,A -85,B 0,C 180,E1 -9429.12,E2 -9429.12} C_VEL
LIN {X 0,Y 433,Z 214.129,A -85,B 0,C 180,E1 -9432.037,E2 -9432.037} C_VEL
LIN {X 0,Y 432.632,Z 220.515,A -85,B 0,C 180,E1 -9433.706,E2 -9433.706} C_VEL
LIN {X 0,Y 434.452,Z 232.707,A -85,B 0,C 180,E1 -9434.142,E2 -9434.142} C_VEL
LIN {X 0,Y 435.002,Z 241.68,A -85,B 0,C 180,E1 -9434.538,E2 -9434.538} C_VEL
LIN {X 0,Y 434.451,Z 254.586,A -85,B 0,C 180,E1 -9435.238,E2 -9435.238} C_VEL
LIN {X 0,Y 433.799,Z 266.118,A -85,B 0,C 180,E1 -9436.066,E2 -9436.066} C_VEL
LIN {X 0,Y 433.119,Z 277.473,A -85,B 0,C 180,E1 -9437.107,E2 -9437.107} C_VEL
LIN {X 0,Y 432.651,Z 287.639,A -85,B 0,C 180,E1 -9438.283,E2 -9438.283} C_VEL
LIN {X 0,Y 432.008,Z 297.418,A -85,B 0,C 180,E1 -9439.69,E2 -9439.69} C_VEL
LIN {X 0,Y 431.68,Z 305.186,A -85,B 0,C 180,E1 -9441.101,E2 -9441.101} C_VEL
LIN {X 0,Y 431.439,Z 311.394,A -85,B 0,C 180,E1 -9442.511,E2 -9442.511} C_VEL
LIN {X 0,Y 431.275,Z 316.651,A -85,B 0,C 180,E1 -9444.032,E2 -9444.032} C_VEL
LIN {X 0,Y 431.288,Z 320.04,A -85,B 0,C 180,E1 -9445.325,E2 -9445.325} C_VEL
LIN {X 0,Y 431.228,Z 321.953,A -85,B 0,C 180,E1 -9446.261,E2 -9446.261} C_VEL
LIN {X 0,Y 431.318,Z 323.384,A -85,B 0,C 180,E1 -9447.197,E2 -9447.197} C_VEL
LIN {X 0,Y 431.265,Z 324.396,A -85,B 0,C 180,E1 -9448.131,E2 -9448.131} C_VEL
LIN {X 0,Y 431.252,Z 325.002,A -85,B 0,C 180,E1 -9449.065,E2 -9449.065} C_VEL
LIN {X 0,Y 431.287,Z 325.148,A -85,B 0,C 180,E1 -9449.999,E2 -9449.999} C_VEL
LIN {X 0,Y 431.294,Z 324.881,A -85,B 0,C 180,E1 -9450.932,E2 -9450.932} C_VEL
LIN {X 0,Y 431.285,Z 324.211,A -85,B 0,C 180,E1 -9451.866,E2 -9451.866} C_VEL
LIN {X 0,Y 431.321,Z 323.088,A -85,B 0,C 180,E1 -9452.8,E2 -9452.8} C_VEL
LIN {X 0,Y 431.247,Z 320.565,A -85,B 0,C 180,E1 -9454.204,E2 -9454.204} C_VEL
LIN {X 0,Y 431.307,Z 316.972,A -85,B 0,C 180,E1 -9455.609,E2 -9455.609} C_VEL
LIN {X 0,Y 431.412,Z 312.204,A -85,B 0,C 180,E1 -9457.016,E2 -9457.016} C_VEL
LIN {X 0,Y 431.603,Z 306.113,A -85,B 0,C 180,E1 -9458.426,E2 -9458.426} C_VEL
LIN {X 0,Y 431.857,Z 298.458,A -85,B 0,C 180,E1 -9459.837,E2 -9459.837} C_VEL
LIN {X 0,Y 432.258,Z 290.546,A -85,B 0,C 180,E1 -9461.012,E2 -9461.012} C_VEL
LIN {X 0,Y 432.701,Z 280.83,A -85,B 0,C 180,E1 -9462.188,E2 -9462.188} C_VEL
LIN {X 0,Y 433.131,Z 271.288,A -85,B 0,C 180,E1 -9463.129,E2 -9463.129} C_VEL
LIN {X 0,Y 433.661,Z 261.189,A -85,B 0,C 180,E1 -9463.936,E2 -9463.936} C_VEL
LIN {X 0,Y 434.073,Z 249.771,A -85,B 0,C 180,E1 -9464.652,E2 -9464.652} C_VEL
LIN {X 0,Y 434.258,Z 237.884,A -85,B 0,C 180,E1 -9465.216,E2 -9465.216} C_VEL
LIN {X 0,Y 432.81,Z 224.802,A -85,B 0,C 180,E1 -9465.679,E2 -9465.679} C_VEL
LIN {X 0,Y 432.314,Z 220.436,A -85,B 0,C 180,E1 -9465.799,E2 -9465.799} C_VEL
LIN {X 0,Y 433.085,Z 206.319,A -85,B 0,C 180,E1 -9469.354,E2 -9469.354} C_VEL
LIN {X 0,Y 433.976,Z 192.595,A -85,B 0,C 180,E1 -9472.87,E2 -9472.87} C_VEL
LIN {X 0,Y 435.032,Z 179.206,A -85,B 0,C 180,E1 -9476.374,E2 -9476.374} C_VEL
LIN {X 0,Y 435.301,Z 175.437,A -85,B 0,C 180,E1 -9477.379,E2 -9477.379} C_VEL
LIN {X 0,Y 434.521,Z 169.581,A -85,B 0,C 180,E1 -9479.025,E2 -9479.025} C_VEL
LIN {X 0,Y 432.321,Z 158.636,A -85,B 0,C 180,E1 -9482.292,E2 -9482.292} C_VEL
LIN {X 0,Y 432.335,Z 158.634,A -85,B 0,C 180,E1 -9484.675,E2 -9484.675} C_VEL
LIN {X 0,Y 432.333,Z 158.632,A -85,B 0,C 180,E1 -9488.148,E2 -9488.148} C_VEL
LIN {X 0,Y 432.315,Z 158.631,A -85,B 0,C 180,E1 -9491.599,E2 -9491.599} C_VEL
LIN {X 0,Y 432.324,Z 158.636,A -85,B 0,C 180,E1 -9494.346,E2 -9494.346} C_VEL
LIN {X 0,Y 432.356,Z 158.63,A -85,B 0,C 180,E1 -9497.008,E2 -9497.008} C_VEL
LIN {X 0,Y 432.348,Z 158.63,A -85,B 0,C 180,E1 -9499.815,E2 -9499.815} C_VEL
LIN {X 0,Y 432.295,Z 158.635,A -85,B 0,C 180,E1 -9503.021,E2 -9503.021} C_VEL
LIN {X 0,Y 432.347,Z 158.633,A -85,B 0,C 180,E1 -9505.995,E2 -9505.995} C_VEL
LIN {X 0,Y 432.383,Z 158.627,A -85,B 0,C 180,E1 -9509.743,E2 -9509.743} C_VEL
LIN {X 0,Y 432.387,Z 158.625,A -85,B 0,C 180,E1 -9513.371,E2 -9513.371} C_VEL
LIN {X 0,Y 432.356,Z 158.631,A -85,B 0,C 180,E1 -9516.022,E2 -9516.022} C_VEL
LIN {X 0,Y 432.336,Z 158.631,A -85,B 0,C 180,E1 -9519.045,E2 -9519.045} C_VEL
LIN {X 0,Y 432.364,Z 158.628,A -85,B 0,C 180,E1 -9522.01,E2 -9522.01} C_VEL
LIN {X 0,Y 432.381,Z 158.627,A -85,B 0,C 180,E1 -9524.926,E2 -9524.926} C_VEL
LIN {X 0,Y 432.465,Z 158.616,A -85,B 0,C 180,E1 -9527.803,E2 -9527.803} C_VEL
LIN {X 0,Y 432.476,Z 158.614,A -85,B 0,C 180,E1 -9531.59,E2 -9531.59} C_VEL
LIN {X 0,Y 432.586,Z 158.6,A -85,B 0,C 180,E1 -9534.406,E2 -9534.406} C_VEL
LIN {X 0,Y 432.591,Z 158.599,A -85,B 0,C 180,E1 -9538.138,E2 -9538.138} C_VEL
LIN {X 0,Y 432.717,Z 158.583,A -85,B 0,C 180,E1 -9540,E2 -9540} C_VEL
LIN {X 0,Y 432.573,Z 158.604,A -85,B 0,C 180,E1 -9542.794,E2 -9542.794} C_VEL
LIN {X 0,Y 432.557,Z 158.606,A -85,B 0,C 180,E1 -9546.53,E2 -9546.53} C_VEL
LIN {X 0,Y 432.431,Z 158.62,A -85,B 0,C 180,E1 -9549.353,E2 -9549.353} C_VEL
LIN {X 0,Y 432.43,Z 158.622,A -85,B 0,C 180,E1 -9552.812,E2 -9552.812} C_VEL
LIN {X 0,Y 432.398,Z 158.626,A -85,B 0,C 180,E1 -9556.48,E2 -9556.48} C_VEL
LIN {X 0,Y 432.366,Z 158.63,A -85,B 0,C 180,E1 -9559.959,E2 -9559.959} C_VEL
LIN {X 0,Y 432.313,Z 158.635,A -85,B 0,C 180,E1 -9562.965,E2 -9562.965} C_VEL
LIN {X 0,Y 432.327,Z 158.632,A -85,B 0,C 180,E1 -9565.003,E2 -9565.003} C_VEL
LIN {X 0,Y 432.334,Z 158.634,A -85,B 0,C 180,E1 -9568.127,E2 -9568.127} C_VEL
LIN {X 0,Y 432.309,Z 158.635,A -85,B 0,C 180,E1 -9571.347,E2 -9571.347} C_VEL
LIN {X 0,Y 432.329,Z 158.632,A -85,B 0,C 180,E1 -9574.678,E2 -9574.678} C_VEL
LIN {X 0,Y 432.336,Z 158.632,A -85,B 0,C 180,E1 -9578.15,E2 -9578.15} C_VEL
LIN {X 0,Y 432.322,Z 158.636,A -85,B 0,C 180,E1 -9581.603,E2 -9581.603} C_VEL
LIN {X 0,Y 432.331,Z 158.632,A -85,B 0,C 180,E1 -9584.348,E2 -9584.348} C_VEL
LIN {X 0,Y 432.315,Z 158.635,A -85,B 0,C 180,E1 -9587.016,E2 -9587.016} C_VEL
LIN {X 0,Y 432.325,Z 158.634,A -85,B 0,C 180,E1 -9589.822,E2 -9589.822} C_VEL
LIN {X 0,Y 432.297,Z 158.637,A -85,B 0,C 180,E1 -9593.023,E2 -9593.023} C_VEL
LIN {X 0,Y 432.352,Z 158.629,A -85,B 0,C 180,E1 -9595.998,E2 -9595.998} C_VEL
LIN {X 0,Y 432.39,Z 158.625,A -85,B 0,C 180,E1 -9599.746,E2 -9599.746} C_VEL
LIN {X 0,Y 432.38,Z 158.628,A -85,B 0,C 180,E1 -9602.93,E2 -9602.93} C_VEL
LIN {X 0,Y 432.361,Z 158.626,A -85,B 0,C 180,E1 -9606.025,E2 -9606.025} C_VEL
LIN {X 0,Y 432.347,Z 158.63,A -85,B 0,C 180,E1 -9609.048,E2 -9609.048} C_VEL
LIN {X 0,Y 432.376,Z 158.628,A -85,B 0,C 180,E1 -9612.013,E2 -9612.013} C_VEL
LIN {X 0,Y 432.392,Z 158.626,A -85,B 0,C 180,E1 -9614.928,E2 -9614.928} C_VEL
LIN {X 0,Y 432.458,Z 158.615,A -85,B 0,C 180,E1 -9617.805,E2 -9617.805} C_VEL
LIN {X 0,Y 432.492,Z 158.612,A -85,B 0,C 180,E1 -9621.592,E2 -9621.592} C_VEL
LIN {X 0,Y 432.599,Z 158.599,A -85,B 0,C 180,E1 -9624.408,E2 -9624.408} C_VEL
LIN {X 0,Y 432.605,Z 158.6,A -85,B 0,C 180,E1 -9628.14,E2 -9628.14} C_VEL
LIN {X 0,Y 432.64,Z 158.596,A -85,B 0,C 180,E1 -9630.001,E2 -9630.001} C_VEL
LIN {X 0,Y 432.585,Z 158.599,A -85,B 0,C 180,E1 -9632.795,E2 -9632.795} C_VEL
LIN {X 0,Y 432.468,Z 158.614,A -85,B 0,C 180,E1 -9635.051,E2 -9635.051} C_VEL
LIN {X 0,Y 431.912,Z 158.685,A -85,B 0,C 180,E1 -9635.83,E2 -9635.83} C_VEL
LIN {X 0,Y 429.065,Z 159.04,A -85,B 0,C 180,E1 -9637.095,E2 -9637.095} C_VEL
LIN {X 0,Y 426.577,Z 159.351,A -85,B 0,C 180,E1 -9638.116,E2 -9638.116} C_VEL
LIN {X 0,Y 425.495,Z 159.483,A -85,B 0,C 180,E1 -9638.906,E2 -9638.906} C_VEL
LIN {X 0,Y 425.404,Z 159.493,A -85,B 0,C 180,E1 -9639.174,E2 -9639.174} C_VEL
LIN {X 0,Y 425.397,Z 159.494,A -85,B 0,C 180,E1 -9642.905,E2 -9642.905} C_VEL
LIN {X 0,Y 425.365,Z 159.499,A -85,B 0,C 180,E1 -9646.606,E2 -9646.606} C_VEL
LIN {X 0,Y 425.333,Z 159.505,A -85,B 0,C 180,E1 -9649.637,E2 -9649.637} C_VEL
LIN {X 0,Y 425.291,Z 159.508,A -85,B 0,C 180,E1 -9652.34,E2 -9652.34} C_VEL
LIN {X 0,Y 425.263,Z 159.513,A -85,B 0,C 180,E1 -9655.449,E2 -9655.449} C_VEL
LIN {X 0,Y 425.311,Z 159.509,A -85,B 0,C 180,E1 -9658.861,E2 -9658.861} C_VEL
LIN {X 0,Y 425.269,Z 159.511,A -85,B 0,C 180,E1 -9661.928,E2 -9661.928} C_VEL
LIN {X 0,Y 425.301,Z 159.508,A -85,B 0,C 180,E1 -9665.337,E2 -9665.337} C_VEL
LIN {X 0,Y 425.28,Z 159.512,A -85,B 0,C 180,E1 -9668.902,E2 -9668.902} C_VEL
LIN {X 0,Y 425.265,Z 159.513,A -85,B 0,C 180,E1 -9672.656,E2 -9672.656} C_VEL
LIN {X 0,Y 425.29,Z 159.509,A -85,B 0,C 180,E1 -9675.284,E2 -9675.284} C_VEL
LIN {X 0,Y 425.278,Z 159.513,A -85,B 0,C 180,E1 -9678.622,E2 -9678.622} C_VEL
LIN {X 0,Y 425.276,Z 159.513,A -85,B 0,C 180,E1 -9682.305,E2 -9682.305} C_VEL
LIN {X 0,Y 425.31,Z 159.509,A -85,B 0,C 180,E1 -9685.818,E2 -9685.818} C_VEL
LIN {X 0,Y 425.373,Z 159.538,A -85,B 0,C 180,E1 -9687.226,E2 -9687.226} C_VEL
LIN {X 0,Y 426.123,Z 164.133,A -85,B 0,C 180,E1 -9689.251,E2 -9689.251} C_VEL
LIN {X 0,Y 426.035,Z 169.26,A -85,B 0,C 180,E1 -9691.42,E2 -9691.42} C_VEL
LIN {X 0,Y 425.76,Z 175.636,A -85,B 0,C 180,E1 -9694.06,E2 -9694.06} C_VEL
LIN {X 0,Y 425.38,Z 183.21,A -85,B 0,C 180,E1 -9697.154,E2 -9697.154} C_VEL
LIN {X 0,Y 425.126,Z 191.375,A -85,B 0,C 180,E1 -9700.444,E2 -9700.444} C_VEL
LIN {X 0,Y 424.863,Z 199.507,A -85,B 0,C 180,E1 -9703.668,E2 -9703.668} C_VEL
LIN {X 0,Y 424.616,Z 208.245,A -85,B 0,C 180,E1 -9707.089,E2 -9707.089} C_VEL
LIN {X 0,Y 424.442,Z 215.341,A -85,B 0,C 180,E1 -9709.837,E2 -9709.837} C_VEL
LIN {X 0,Y 425.756,Z 227.716,A -85,B 0,C 180,E1 -9710.499,E2 -9710.499} C_VEL
LIN {X 0,Y 425.841,Z 234.737,A -85,B 0,C 180,E1 -9710.98,E2 -9710.98} C_VEL
LIN {X 0,Y 425.459,Z 244.283,A -85,B 0,C 180,E1 -9711.809,E2 -9711.809} C_VEL
LIN {X 0,Y 425.121,Z 253.123,A -85,B 0,C 180,E1 -9712.816,E2 -9712.816} C_VEL
LIN {X 0,Y 424.877,Z 260.033,A -85,B 0,C 180,E1 -9713.828,E2 -9713.828} C_VEL
LIN {X 0,Y 424.642,Z 266.318,A -85,B 0,C 180,E1 -9715.015,E2 -9715.015} C_VEL
LIN {X 0,Y 424.568,Z 271.058,A -85,B 0,C 180,E1 -9716.204,E2 -9716.204} C_VEL
LIN {X 0,Y 424.285,Z 275.032,A -85,B 0,C 180,E1 -9717.627,E2 -9717.627} C_VEL
LIN {X 0,Y 424.21,Z 277.358,A -85,B 0,C 180,E1 -9719.051,E2 -9719.051} C_VEL
LIN {X 0,Y 424.225,Z 278.057,A -85,B 0,C 180,E1 -9720,E2 -9720} C_VEL
LIN {X 0,Y 424.273,Z 278.086,A -85,B 0,C 180,E1 -9720.949,E2 -9720.949} C_VEL
LIN {X 0,Y 424.382,Z 277.443,A -85,B 0,C 180,E1 -9721.898,E2 -9721.898} C_VEL
LIN {X 0,Y 424.66,Z 275.199,A -85,B 0,C 180,E1 -9723.321,E2 -9723.321} C_VEL
LIN {X 0,Y 424.845,Z 272.816,A -85,B 0,C 180,E1 -9724.269,E2 -9724.269} C_VEL
LIN {X 0,Y 424.967,Z 269.668,A -85,B 0,C 180,E1 -9725.219,E2 -9725.219} C_VEL
LIN {X 0,Y 425.216,Z 264.517,A -85,B 0,C 180,E1 -9726.406,E2 -9726.406} C_VEL
LIN {X 0,Y 425.672,Z 257.712,A -85,B 0,C 180,E1 -9727.59,E2 -9727.59} C_VEL
LIN {X 0,Y 426.23,Z 249.795,A -85,B 0,C 180,E1 -9728.654,E2 -9728.654} C_VEL
LIN {X 0,Y 426.86,Z 240.723,A -85,B 0,C 180,E1 -9729.596,E2 -9729.596} C_VEL
LIN {X 0,Y 427.224,Z 232.03,A -85,B 0,C 180,E1 -9730.306,E2 -9730.306} C_VEL
LIN {X 0,Y 425.939,Z 222.207,A -85,B 0,C 180,E1 -9730.998,E2 -9730.998} C_VEL
LIN {X 0,Y 424.837,Z 216.348,A -85,B 0,C 180,E1 -9731.36,E2 -9731.36} C_VEL
LIN {X 0,Y 425.188,Z 207.85,A -85,B 0,C 180,E1 -9734.845,E2 -9734.845} C_VEL
LIN {X 0,Y 425.57,Z 199.692,A -85,B 0,C 180,E1 -9738.287,E2 -9738.287} C_VEL
LIN {X 0,Y 426.058,Z 191.716,A -85,B 0,C 180,E1 -9741.786,E2 -9741.786} C_VEL
LIN {X 0,Y 426.653,Z 183.92,A -85,B 0,C 180,E1 -9745.359,E2 -9745.359} C_VEL
LIN {X 0,Y 427.433,Z 177.508,A -85,B 0,C 180,E1 -9748.479,E2 -9748.479} C_VEL
LIN {X 0,Y 427.777,Z 173.465,A -85,B 0,C 180,E1 -9750.618,E2 -9750.618} C_VEL
LIN {X 0,Y 427.392,Z 169.512,A -85,B 0,C 180,E1 -9753.002,E2 -9753.002} C_VEL
LIN {X 0,Y 426.777,Z 166.396,A -85,B 0,C 180,E1 -9755.196,E2 -9755.196} C_VEL
LIN {X 0,Y 426.205,Z 163.438,A -85,B 0,C 180,E1 -9757.672,E2 -9757.672} C_VEL
LIN {X 0,Y 425.709,Z 161.272,A -85,B 0,C 180,E1 -9760.08,E2 -9760.08} C_VEL
LIN {X 0,Y 425.297,Z 159.558,A -85,B 0,C 180,E1 -9763.355,E2 -9763.355} C_VEL
LIN {X 0,Y 425.285,Z 159.511,A -85,B 0,C 180,E1 -9766.826,E2 -9766.826} C_VEL
LIN {X 0,Y 425.712,Z 161.067,A -85,B 0,C 180,E1 -9769.92,E2 -9769.92} C_VEL
LIN {X 0,Y 426.284,Z 163.522,A -85,B 0,C 180,E1 -9772.409,E2 -9772.409} C_VEL
LIN {X 0,Y 427.251,Z 167.652,A -85,B 0,C 180,E1 -9775.333,E2 -9775.333} C_VEL
LIN {X 0,Y 428.253,Z 172.093,A -85,B 0,C 180,E1 -9777.766,E2 -9777.766} C_VEL
LIN {X 0,Y 429.306,Z 177.364,A -85,B 0,C 180,E1 -9780.186,E2 -9780.186} C_VEL
LIN {X 0,Y 429.873,Z 181.127,A -85,B 0,C 180,E1 -9781.697,E2 -9781.697} C_VEL
LIN {X 0,Y 429.345,Z 185.613,A -85,B 0,C 180,E1 -9783.245,E2 -9783.245} C_VEL
LIN {X 0,Y 427.931,Z 195.264,A -85,B 0,C 180,E1 -9786.272,E2 -9786.272} C_VEL
LIN {X 0,Y 426.617,Z 207.655,A -85,B 0,C 180,E1 -9789.886,E2 -9789.886} C_VEL
LIN {X 0,Y 425.644,Z 220.466,A -85,B 0,C 180,E1 -9793.378,E2 -9793.378} C_VEL
LIN {X 0,Y 427.657,Z 233.17,A -85,B 0,C 180,E1 -9793.868,E2 -9793.868} C_VEL
LIN {X 0,Y 428.141,Z 243.397,A -85,B 0,C 180,E1 -9794.345,E2 -9794.345} C_VEL
LIN {X 0,Y 427.611,Z 254.882,A -85,B 0,C 180,E1 -9794.996,E2 -9794.996} C_VEL
LIN {X 0,Y 426.924,Z 266.221,A -85,B 0,C 180,E1 -9795.837,E2 -9795.837} C_VEL
LIN {X 0,Y 426.168,Z 277.531,A -85,B 0,C 180,E1 -9796.899,E2 -9796.899} C_VEL
LIN {X 0,Y 425.671,Z 287.544,A -85,B 0,C 180,E1 -9798.088,E2 -9798.088} C_VEL
LIN {X 0,Y 424.988,Z 297.264,A -85,B 0,C 180,E1 -9799.518,E2 -9799.518} C_VEL
LIN {X 0,Y 424.617,Z 304.967,A -85,B 0,C 180,E1 -9800.952,E2 -9800.952} C_VEL
LIN {X 0,Y 424.366,Z 311.141,A -85,B 0,C 180,E1 -9802.385,E2 -9802.385} C_VEL
LIN {X 0,Y 424.225,Z 315.73,A -85,B 0,C 180,E1 -9803.723,E2 -9803.723} C_VEL
LIN {X 0,Y 424.218,Z 319.729,A -85,B 0,C 180,E1 -9805.247,E2 -9805.247} C_VEL
LIN {X 0,Y 424.136,Z 321.613,A -85,B 0,C 180,E1 -9806.198,E2 -9806.198} C_VEL
LIN {X 0,Y 424.227,Z 323.028,A -85,B 0,C 180,E1 -9807.15,E2 -9807.15} C_VEL
LIN {X 0,Y 424.188,Z 324.028,A -85,B 0,C 180,E1 -9808.1,E2 -9808.1} C_VEL
LIN {X 0,Y 424.167,Z 324.61,A -85,B 0,C 180,E1 -9809.049,E2 -9809.049} C_VEL
LIN {X 0,Y 424.211,Z 324.734,A -85,B 0,C 180,E1 -9809.999,E2 -9809.999} C_VEL
LIN {X 0,Y 424.206,Z 324.45,A -85,B 0,C 180,E1 -9810.948,E2 -9810.948} C_VEL
LIN {X 0,Y 424.207,Z 323.76,A -85,B 0,C 180,E1 -9811.897,E2 -9811.897} C_VEL
LIN {X 0,Y 424.249,Z 322.599,A -85,B 0,C 180,E1 -9812.847,E2 -9812.847} C_VEL
LIN {X 0,Y 424.166,Z 320.028,A -85,B 0,C 180,E1 -9814.274,E2 -9814.274} C_VEL
LIN {X 0,Y 424.21,Z 316.382,A -85,B 0,C 180,E1 -9815.703,E2 -9815.703} C_VEL
LIN {X 0,Y 424.337,Z 311.556,A -85,B 0,C 180,E1 -9817.134,E2 -9817.134} C_VEL
LIN {X 0,Y 424.521,Z 305.394,A -85,B 0,C 180,E1 -9818.567,E2 -9818.567} C_VEL
LIN {X 0,Y 424.798,Z 297.614,A -85,B 0,C 180,E1 -9820.002,E2 -9820.002} C_VEL
LIN {X 0,Y 425.216,Z 289.593,A -85,B 0,C 180,E1 -9821.197,E2 -9821.197} C_VEL
LIN {X 0,Y 425.691,Z 279.753,A -85,B 0,C 180,E1 -9822.392,E2 -9822.392} C_VEL
LIN {X 0,Y 426.126,Z 270.036,A -85,B 0,C 180,E1 -9823.348,E2 -9823.348} C_VEL
LIN {X 0,Y 426.756,Z 257.72,A -85,B 0,C 180,E1 -9824.3,E2 -9824.3} C_VEL
LIN {X 0,Y 427.224,Z 245.62,A -85,B 0,C 180,E1 -9825.015,E2 -9825.015} C_VEL
LIN {X 0,Y 427.17,Z 237.941,A -85,B 0,C 180,E1 -9825.368,E2 -9825.368} C_VEL
LIN {X 0,Y 425.805,Z 225.231,A -85,B 0,C 180,E1 -9825.832,E2 -9825.832} C_VEL
LIN {X 0,Y 425.287,Z 220.377,A -85,B 0,C 180,E1 -9825.975,E2 -9825.975} C_VEL
LIN {X 0,Y 426.078,Z 206.267,A -85,B 0,C 180,E1 -9829.605,E2 -9829.605} C_VEL
LIN {X 0,Y 427.084,Z 192.313,A -85,B 0,C 180,E1 -9833.26,E2 -9833.26} C_VEL
LIN {X 0,Y 428.194,Z 178.912,A -85,B 0,C 180,E1 -9836.829,E2 -9836.829} C_VEL
LIN {X 0,Y 428.24,Z 174.823,A -85,B 0,C 180,E1 -9837.958,E2 -9837.958} C_VEL
LIN {X 0,Y 426.47,Z 165.431,A -85,B 0,C 180,E1 -9840.719,E2 -9840.719} C_VEL
LIN {X 0,Y 425.276,Z 159.513,A -85,B 0,C 180,E1 -9842.561,E2 -9842.561} C_VEL
LIN {X 0,Y 425.294,Z 159.512,A -85,B 0,C 180,E1 -9845.334,E2 -9845.334} C_VEL
LIN {X 0,Y 425.287,Z 159.512,A -85,B 0,C 180,E1 -9848.897,E2 -9848.897} C_VEL
LIN {X 0,Y 425.273,Z 159.509,A -85,B 0,C 180,E1 -9851.955,E2 -9851.955} C_VEL
LIN {X 0,Y 425.304,Z 159.507,A -85,B 0,C 180,E1 -9855.278,E2 -9855.278} C_VEL
LIN {X 0,Y 425.3,Z 159.509,A -85,B 0,C 180,E1 -9858.624,E2 -9858.624} C_VEL
LIN {X 0,Y 425.31,Z 159.506,A -85,B 0,C 180,E1 -9861.102,E2 -9861.102} C_VEL
LIN {X 0,Y 425.286,Z 159.508,A -85,B 0,C 180,E1 -9864.663,E2 -9864.663} C_VEL
LIN {X 0,Y 425.255,Z 159.515,A -85,B 0,C 180,E1 -9868.072,E2 -9868.072} C_VEL
LIN {X 0,Y 425.325,Z 159.506,A -85,B 0,C 180,E1 -9871.367,E2 -9871.367} C_VEL
LIN {X 0,Y 425.28,Z 159.51,A -85,B 0,C 180,E1 -9874.554,E2 -9874.554} C_VEL
LIN {X 0,Y 425.274,Z 159.514,A -85,B 0,C 180,E1 -9877.66,E2 -9877.66} C_VEL
LIN {X 0,Y 425.348,Z 159.501,A -85,B 0,C 180,E1 -9880.703,E2 -9880.703} C_VEL
LIN {X 0,Y 425.374,Z 159.499,A -85,B 0,C 180,E1 -9883.688,E2 -9883.688} C_VEL
LIN {X 0,Y 425.415,Z 159.497,A -85,B 0,C 180,E1 -9887.598,E2 -9887.598} C_VEL
LIN {X 0,Y 425.427,Z 159.493,A -85,B 0,C 180,E1 -9891.45,E2 -9891.45} C_VEL
LIN {X 0,Y 425.543,Z 159.477,A -85,B 0,C 180,E1 -9894.313,E2 -9894.313} C_VEL
LIN {X 0,Y 425.561,Z 159.475,A -85,B 0,C 180,E1 -9898.107,E2 -9898.107} C_VEL
LIN {X 0,Y 425.686,Z 159.458,A -85,B 0,C 180,E1 -9900,E2 -9900} C_VEL
LIN {X 0,Y 425.527,Z 159.483,A -85,B 0,C 180,E1 -9902.84,E2 -9902.84} C_VEL
LIN {X 0,Y 425.516,Z 159.483,A -85,B 0,C 180,E1 -9906.639,E2 -9906.639} C_VEL
LIN {X 0,Y 425.39,Z 159.497,A -85,B 0,C 180,E1 -9909.51,E2 -9909.51} C_VEL
LIN {X 0,Y 425.389,Z 159.498,A -85,B 0,C 180,E1 -9912.911,E2 -9912.911} C_VEL
LIN {X 0,Y 425.347,Z 159.503,A -85,B 0,C 180,E1 -9916.606,E2 -9916.606} C_VEL
LIN {X 0,Y 425.348,Z 159.502,A -85,B 0,C 180,E1 -9919.649,E2 -9919.649} C_VEL
LIN {X 0,Y 425.297,Z 159.508,A -85,B 0,C 180,E1 -9923.366,E2 -9923.366} C_VEL
LIN {X 0,Y 425.288,Z 159.51,A -85,B 0,C 180,E1 -9926.499,E2 -9926.499} C_VEL
LIN {X 0,Y 425.273,Z 159.513,A -85,B 0,C 180,E1 -9929.721,E2 -9929.721} C_VEL
LIN {X 0,Y 425.27,Z 159.511,A -85,B 0,C 180,E1 -9933.049,E2 -9933.049} C_VEL
LIN {X 0,Y 425.273,Z 159.513,A -85,B 0,C 180,E1 -9935.93,E2 -9935.93} C_VEL
LIN {X 0,Y 425.292,Z 159.507,A -85,B 0,C 180,E1 -9939.046,E2 -9939.046} C_VEL
LIN {X 0,Y 425.267,Z 159.511,A -85,B 0,C 180,E1 -9942.654,E2 -9942.654} C_VEL
LIN {X 0,Y 425.259,Z 159.514,A -85,B 0,C 180,E1 -9946.047,E2 -9946.047} C_VEL
LIN {X 0,Y 425.266,Z 159.512,A -85,B 0,C 180,E1 -9948.623,E2 -9948.623} C_VEL
LIN {X 0,Y 425.288,Z 159.51,A -85,B 0,C 180,E1 -9951.103,E2 -9951.103} C_VEL
LIN {X 0,Y 425.291,Z 159.509,A -85,B 0,C 180,E1 -9954.666,E2 -9954.666} C_VEL
LIN {X 0,Y 425.262,Z 159.512,A -85,B 0,C 180,E1 -9958.075,E2 -9958.075} C_VEL
LIN {X 0,Y 425.332,Z 159.506,A -85,B 0,C 180,E1 -9961.37,E2 -9961.37} C_VEL
LIN {X 0,Y 425.278,Z 159.511,A -85,B 0,C 180,E1 -9964.556,E2 -9964.556} C_VEL
LIN {X 0,Y 425.299,Z 159.511,A -85,B 0,C 180,E1 -9966.636,E2 -9966.636} C_VEL
LIN {X 0,Y 425.326,Z 159.507,A -85,B 0,C 180,E1 -9970.366,E2 -9970.366} C_VEL
LIN {X 0,Y 425.387,Z 159.497,A -85,B 0,C 180,E1 -9973.69,E2 -9973.69} C_VEL
LIN {X 0,Y 425.411,Z 159.492,A -85,B 0,C 180,E1 -9977.6,E2 -9977.6} C_VEL
LIN {X 0,Y 425.442,Z 159.489,A -85,B 0,C 180,E1 -9981.452,E2 -9981.452} C_VEL
LIN {X 0,Y 425.555,Z 159.477,A -85,B 0,C 180,E1 -9984.315,E2 -9984.315} C_VEL
LIN {X 0,Y 425.574,Z 159.476,A -85,B 0,C 180,E1 -9988.109,E2 -9988.109} C_VEL
LIN {X 0,Y 425.592,Z 159.474,A -85,B 0,C 180,E1 -9990.001,E2 -9990.001} C_VEL
LIN {X 0,Y 425.539,Z 159.477,A -85,B 0,C 180,E1 -9992.841,E2 -9992.841} C_VEL
LIN {X 0,Y 425.534,Z 159.479,A -85,B 0,C 180,E1 -9996.64,E2 -9996.64} C_VEL
LIN {X 0,Y 425.404,Z 159.493,A -85,B 0,C 180,E1 -9999.174,E2 -9999.174} C_VEL
LIN {X 0,Y 424.733,Z 159.581,A -85,B 0,C 180,E1 -9999.964,E2 -9999.964} C_VEL
LIN {X 0,Y 421.885,Z 159.933,A -85,B 0,C 180,E1 -10001.247,E2 -10001.247} C_VEL
LIN {X 0,Y 419.469,Z 160.233,A -85,B 0,C 180,E1 -10002.283,E2 -10002.283} C_VEL
LIN {X 0,Y 418.417,Z 160.364,A -85,B 0,C 180,E1 -10003.084,E2 -10003.084} C_VEL
LIN {X 0,Y 418.324,Z 160.377,A -85,B 0,C 180,E1 -10003.355,E2 -10003.355} C_VEL
LIN {X 0,Y 418.317,Z 160.377,A -85,B 0,C 180,E1 -10006.736,E2 -10006.736} C_VEL
LIN {X 0,Y 418.275,Z 160.385,A -85,B 0,C 180,E1 -10009.791,E2 -10009.791} C_VEL
LIN {X 0,Y 418.232,Z 160.388,A -85,B 0,C 180,E1 -10012.738,E2 -10012.738} C_VEL
LIN {X 0,Y 418.222,Z 160.387,A -85,B 0,C 180,E1 -10015.909,E2 -10015.909} C_VEL
LIN {X 0,Y 418.263,Z 160.385,A -85,B 0,C 180,E1 -10019.163,E2 -10019.163} C_VEL
LIN {X 0,Y 418.262,Z 160.385,A -85,B 0,C 180,E1 -10022.845,E2 -10022.845} C_VEL
LIN {X 0,Y 418.245,Z 160.386,A -85,B 0,C 180,E1 -10026.238,E2 -10026.238} C_VEL
LIN {X 0,Y 418.203,Z 160.39,A -85,B 0,C 180,E1 -10029.689,E2 -10029.689} C_VEL
LIN {X 0,Y 418.217,Z 160.393,A -85,B 0,C 180,E1 -10032.319,E2 -10032.319} C_VEL
LIN {X 0,Y 418.241,Z 160.388,A -85,B 0,C 180,E1 -10035.109,E2 -10035.109} C_VEL
LIN {X 0,Y 418.245,Z 160.387,A -85,B 0,C 180,E1 -10037.767,E2 -10037.767} C_VEL
LIN {X 0,Y 418.24,Z 160.385,A -85,B 0,C 180,E1 -10041.557,E2 -10041.557} C_VEL
LIN {X 0,Y 418.263,Z 160.384,A -85,B 0,C 180,E1 -10045.159,E2 -10045.159} C_VEL
LIN {X 0,Y 418.347,Z 160.5,A -85,B 0,C 180,E1 -10047.139,E2 -10047.139} C_VEL
LIN {X 0,Y 419.119,Z 165.372,A -85,B 0,C 180,E1 -10049.314,E2 -10049.314} C_VEL
LIN {X 0,Y 419,Z 170.36,A -85,B 0,C 180,E1 -10051.443,E2 -10051.443} C_VEL
LIN {X 0,Y 418.661,Z 177.973,A -85,B 0,C 180,E1 -10054.642,E2 -10054.642} C_VEL
LIN {X 0,Y 418.31,Z 184.968,A -85,B 0,C 180,E1 -10057.528,E2 -10057.528} C_VEL
LIN {X 0,Y 418.02,Z 193.173,A -85,B 0,C 180,E1 -10060.862,E2 -10060.862} C_VEL
LIN {X 0,Y 417.752,Z 201.943,A -85,B 0,C 180,E1 -10064.385,E2 -10064.385} C_VEL
LIN {X 0,Y 417.518,Z 210.875,A -85,B 0,C 180,E1 -10067.922,E2 -10067.922} C_VEL
LIN {X 0,Y 417.363,Z 215.395,A -85,B 0,C 180,E1 -10069.693,E2 -10069.693} C_VEL
LIN {X 0,Y 418.65,Z 227.308,A -85,B 0,C 180,E1 -10070.336,E2 -10070.336} C_VEL
LIN {X 0,Y 418.826,Z 234.44,A -85,B 0,C 180,E1 -10070.827,E2 -10070.827} C_VEL
LIN {X 0,Y 418.422,Z 244.122,A -85,B 0,C 180,E1 -10071.67,E2 -10071.67} C_VEL
LIN {X 0,Y 418.106,Z 252.614,A -85,B 0,C 180,E1 -10072.637,E2 -10072.637} C_VEL
LIN {X 0,Y 417.818,Z 260.046,A -85,B 0,C 180,E1 -10073.723,E2 -10073.723} C_VEL
LIN {X 0,Y 417.576,Z 266.415,A -85,B 0,C 180,E1 -10074.931,E2 -10074.931} C_VEL
LIN {X 0,Y 417.481,Z 271.233,A -85,B 0,C 180,E1 -10076.139,E2 -10076.139} C_VEL
LIN {X 0,Y 417.21,Z 275.29,A -85,B 0,C 180,E1 -10077.586,E2 -10077.586} C_VEL
LIN {X 0,Y 417.127,Z 277.702,A -85,B 0,C 180,E1 -10079.035,E2 -10079.035} C_VEL
LIN {X 0,Y 417.137,Z 278.456,A -85,B 0,C 180,E1 -10080,E2 -10080} C_VEL
LIN {X 0,Y 417.217,Z 278.539,A -85,B 0,C 180,E1 -10080.965,E2 -10080.965} C_VEL
LIN {X 0,Y 417.332,Z 277.952,A -85,B 0,C 180,E1 -10081.93,E2 -10081.93} C_VEL
LIN {X 0,Y 417.533,Z 276.688,A -85,B 0,C 180,E1 -10082.895,E2 -10082.895} C_VEL
LIN {X 0,Y 417.811,Z 273.481,A -85,B 0,C 180,E1 -10084.341,E2 -10084.341} C_VEL
LIN {X 0,Y 418.095,Z 268.552,A -85,B 0,C 180,E1 -10085.789,E2 -10085.789} C_VEL
LIN {X 0,Y 418.381,Z 263.144,A -85,B 0,C 180,E1 -10086.956,E2 -10086.956} C_VEL
LIN {X 0,Y 418.885,Z 256.702,A -85,B 0,C 180,E1 -10088.03,E2 -10088.03} C_VEL
LIN {X 0,Y 419.565,Z 247.987,A -85,B 0,C 180,E1 -10089.157,E2 -10089.157} C_VEL
LIN {X 0,Y 420.156,Z 239.706,A -85,B 0,C 180,E1 -10089.994,E2 -10089.994} C_VEL
LIN {X 0,Y 420.375,Z 232.401,A -85,B 0,C 180,E1 -10090.597,E2 -10090.597} C_VEL
LIN {X 0,Y 418.913,Z 221.8,A -85,B 0,C 180,E1 -10091.369,E2 -10091.369} C_VEL
LIN {X 0,Y 417.836,Z 216.468,A -85,B 0,C 180,E1 -10091.706,E2 -10091.706} C_VEL
LIN {X 0,Y 418.189,Z 208.384,A -85,B 0,C 180,E1 -10095.099,E2 -10095.099} C_VEL
LIN {X 0,Y 418.568,Z 201.42,A -85,B 0,C 180,E1 -10098.097,E2 -10098.097} C_VEL
LIN {X 0,Y 419.087,Z 193.461,A -85,B 0,C 180,E1 -10101.65,E2 -10101.65} C_VEL
LIN {X 0,Y 419.714,Z 185.728,A -85,B 0,C 180,E1 -10105.28,E2 -10105.28} C_VEL
LIN {X 0,Y 420.535,Z 179.379,A -85,B 0,C 180,E1 -10108.444,E2 -10108.444} C_VEL
LIN {X 0,Y 420.849,Z 176.361,A -85,B 0,C 180,E1 -10110.066,E2 -10110.066} C_VEL
LIN {X 0,Y 420.884,Z 173.716,A -85,B 0,C 180,E1 -10111.611,E2 -10111.611} C_VEL
LIN {X 0,Y 420.18,Z 169.271,A -85,B 0,C 180,E1 -10114.659,E2 -10114.659} C_VEL
LIN {X 0,Y 419.399,Z 165.361,A -85,B 0,C 180,E1 -10118.037,E2 -10118.037} C_VEL
LIN {X 0,Y 418.887,Z 163.12,A -85,B 0,C 180,E1 -10120.973,E2 -10120.973} C_VEL
LIN {X 0,Y 418.632,Z 162,A -85,B 0,C 180,E1 -10123.788,E2 -10123.788} C_VEL
LIN {X 0,Y 418.627,Z 162.044,A -85,B 0,C 180,E1 -10126.502,E2 -10126.502} C_VEL
LIN {X 0,Y 418.907,Z 163.138,A -85,B 0,C 180,E1 -10129.132,E2 -10129.132} C_VEL
LIN {X 0,Y 419.424,Z 165.261,A -85,B 0,C 180,E1 -10131.684,E2 -10131.684} C_VEL
LIN {X 0,Y 420.18,Z 168.36,A -85,B 0,C 180,E1 -10134.166,E2 -10134.166} C_VEL
LIN {X 0,Y 421.308,Z 173.298,A -85,B 0,C 180,E1 -10137.169,E2 -10137.169} C_VEL
LIN {X 0,Y 422.447,Z 178.915,A -85,B 0,C 180,E1 -10139.894,E2 -10139.894} C_VEL
LIN {X 0,Y 423.083,Z 183.245,A -85,B 0,C 180,E1 -10141.692,E2 -10141.692} C_VEL
LIN {X 0,Y 422.199,Z 189.221,A -85,B 0,C 180,E1 -10143.768,E2 -10143.768} C_VEL
LIN {X 0,Y 420.498,Z 200.726,A -85,B 0,C 180,E1 -10147.391,E2 -10147.391} C_VEL
LIN {X 0,Y 419.465,Z 211.059,A -85,B 0,C 180,E1 -10150.42,E2 -10150.42} C_VEL
LIN {X 0,Y 418.714,Z 220.445,A -85,B 0,C 180,E1 -10153.034,E2 -10153.034} C_VEL
LIN {X 0,Y 420.901,Z 233.876,A -85,B 0,C 180,E1 -10153.586,E2 -10153.586} C_VEL
LIN {X 0,Y 421.366,Z 244.096,A -85,B 0,C 180,E1 -10154.087,E2 -10154.087} C_VEL
LIN {X 0,Y 420.786,Z 255.283,A -85,B 0,C 180,E1 -10154.747,E2 -10154.747} C_VEL
LIN {X 0,Y 420.046,Z 266.283,A -85,B 0,C 180,E1 -10155.587,E2 -10155.587} C_VEL
LIN {X 0,Y 419.288,Z 277.058,A -85,B 0,C 180,E1 -10156.622,E2 -10156.622} C_VEL
LIN {X 0,Y 418.779,Z 285.707,A -85,B 0,C 180,E1 -10157.643,E2 -10157.643} C_VEL
LIN {X 0,Y 418.208,Z 294.174,A -85,B 0,C 180,E1 -10158.856,E2 -10158.856} C_VEL
LIN {X 0,Y 417.708,Z 302.416,A -85,B 0,C 180,E1 -10160.312,E2 -10160.312} C_VEL
LIN {X 0,Y 417.414,Z 309.052,A -85,B 0,C 180,E1 -10161.77,E2 -10161.77} C_VEL
LIN {X 0,Y 417.231,Z 314.293,A -85,B 0,C 180,E1 -10163.227,E2 -10163.227} C_VEL
LIN {X 0,Y 417.14,Z 318.327,A -85,B 0,C 180,E1 -10164.682,E2 -10164.682} C_VEL
LIN {X 0,Y 417.049,Z 321.278,A -85,B 0,C 180,E1 -10166.133,E2 -10166.133} C_VEL
LIN {X 0,Y 417.123,Z 322.679,A -85,B 0,C 180,E1 -10167.101,E2 -10167.101} C_VEL
LIN {X 0,Y 417.114,Z 323.665,A -85,B 0,C 180,E1 -10168.067,E2 -10168.067} C_VEL
LIN {X 0,Y 417.085,Z 324.211,A -85,B 0,C 180,E1 -10169.033,E2 -10169.033} C_VEL
LIN {X 0,Y 417.124,Z 324.315,A -85,B 0,C 180,E1 -10169.998,E2 -10169.998} C_VEL
LIN {X 0,Y 417.122,Z 324.013,A -85,B 0,C 180,E1 -10170.964,E2 -10170.964} C_VEL
LIN {X 0,Y 417.132,Z 323.291,A -85,B 0,C 180,E1 -10171.929,E2 -10171.929} C_VEL
LIN {X 0,Y 417.178,Z 322.098,A -85,B 0,C 180,E1 -10172.895,E2 -10172.895} C_VEL
LIN {X 0,Y 417.091,Z 319.479,A -85,B 0,C 180,E1 -10174.347,E2 -10174.347} C_VEL
LIN {X 0,Y 417.126,Z 315.777,A -85,B 0,C 180,E1 -10175.8,E2 -10175.8} C_VEL
LIN {X 0,Y 417.263,Z 310.887,A -85,B 0,C 180,E1 -10177.256,E2 -10177.256} C_VEL
LIN {X 0,Y 417.45,Z 304.651,A -85,B 0,C 180,E1 -10178.713,E2 -10178.713} C_VEL
LIN {X 0,Y 417.735,Z 296.734,A -85,B 0,C 180,E1 -10180.173,E2 -10180.173} C_VEL
LIN {X 0,Y 418.203,Z 288.607,A -85,B 0,C 180,E1 -10181.387,E2 -10181.387} C_VEL
LIN {X 0,Y 418.644,Z 279.7,A -85,B 0,C 180,E1 -10182.481,E2 -10182.481} C_VEL
LIN {X 0,Y 419.081,Z 270.317,A -85,B 0,C 180,E1 -10183.427,E2 -10183.427} C_VEL
LIN {X 0,Y 419.675,Z 259.551,A -85,B 0,C 180,E1 -10184.299,E2 -10184.299} C_VEL
LIN {X 0,Y 420.187,Z 246.946,A -85,B 0,C 180,E1 -10185.086,E2 -10185.086} C_VEL
LIN {X 0,Y 420.164,Z 238.626,A -85,B 0,C 180,E1 -10185.49,E2 -10185.49} C_VEL
LIN {X 0,Y 418.724,Z 225.173,A -85,B 0,C 180,E1 -10185.998,E2 -10185.998} C_VEL
LIN {X 0,Y 418.223,Z 220.325,A -85,B 0,C 180,E1 -10186.158,E2 -10186.158} C_VEL
LIN {X 0,Y 419.019,Z 207.183,A -85,B 0,C 180,E1 -10189.598,E2 -10189.598} C_VEL
LIN {X 0,Y 420.045,Z 193.384,A -85,B 0,C 180,E1 -10193.275,E2 -10193.275} C_VEL
LIN {X 0,Y 421.158,Z 180.524,A -85,B 0,C 180,E1 -10196.777,E2 -10196.777} C_VEL
LIN {X 0,Y 421.306,Z 176.66,A -85,B 0,C 180,E1 -10197.856,E2 -10197.856} C_VEL
LIN {X 0,Y 419.946,Z 168.962,A -85,B 0,C 180,E1 -10200.135,E2 -10200.135} C_VEL
LIN {X 0,Y 418.244,Z 160.389,A -85,B 0,C 180,E1 -10202.841,E2 -10202.841} C_VEL
LIN {X 0,Y 418.24,Z 160.392,A -85,B 0,C 180,E1 -10206.022,E2 -10206.022} C_VEL
LIN {X 0,Y 418.235,Z 160.386,A -85,B 0,C 180,E1 -10209.681,E2 -10209.681} C_VEL
LIN {X 0,Y 418.215,Z 160.391,A -85,B 0,C 180,E1 -10212.319,E2 -10212.319} C_VEL
LIN {X 0,Y 418.249,Z 160.386,A -85,B 0,C 180,E1 -10215.11,E2 -10215.11} C_VEL
LIN {X 0,Y 418.283,Z 160.382,A -85,B 0,C 180,E1 -10217.772,E2 -10217.772} C_VEL
LIN {X 0,Y 418.252,Z 160.385,A -85,B 0,C 180,E1 -10221.558,E2 -10221.558} C_VEL
LIN {X 0,Y 418.247,Z 160.384,A -85,B 0,C 180,E1 -10225.158,E2 -10225.158} C_VEL
LIN {X 0,Y 418.234,Z 160.388,A -85,B 0,C 180,E1 -10227.471,E2 -10227.471} C_VEL
LIN {X 0,Y 418.264,Z 160.384,A -85,B 0,C 180,E1 -10230.892,E2 -10230.892} C_VEL
LIN {X 0,Y 418.256,Z 160.388,A -85,B 0,C 180,E1 -10234.095,E2 -10234.095} C_VEL
LIN {X 0,Y 418.218,Z 160.389,A -85,B 0,C 180,E1 -10237.263,E2 -10237.263} C_VEL
LIN {X 0,Y 418.269,Z 160.383,A -85,B 0,C 180,E1 -10240.363,E2 -10240.363} C_VEL
LIN {X 0,Y 418.303,Z 160.38,A -85,B 0,C 180,E1 -10243.404,E2 -10243.404} C_VEL
LIN {X 0,Y 418.341,Z 160.374,A -85,B 0,C 180,E1 -10246.993,E2 -10246.993} C_VEL
LIN {X 0,Y 418.326,Z 160.374,A -85,B 0,C 180,E1 -10250.328,E2 -10250.328} C_VEL
LIN {X 0,Y 418.48,Z 160.359,A -85,B 0,C 180,E1 -10253.249,E2 -10253.249} C_VEL
LIN {X 0,Y 418.331,Z 160.377,A -85,B 0,C 180,E1 -10255.181,E2 -10255.181} C_VEL
LIN {X 0,Y 418.53,Z 160.35,A -85,B 0,C 180,E1 -10258.075,E2 -10258.075} C_VEL
LIN {X 0,Y 418.656,Z 160.334,A -85,B 0,C 180,E1 -10260,E2 -10260} C_VEL
LIN {X 0,Y 418.482,Z 160.36,A -85,B 0,C 180,E1 -10262.888,E2 -10262.888} C_VEL
LIN {X 0,Y 418.478,Z 160.359,A -85,B 0,C 180,E1 -10266.751,E2 -10266.751} C_VEL
LIN {X 0,Y 418.346,Z 160.374,A -85,B 0,C 180,E1 -10269.671,E2 -10269.671} C_VEL
LIN {X 0,Y 418.341,Z 160.375,A -85,B 0,C 180,E1 -10273.007,E2 -10273.007} C_VEL
LIN {X 0,Y 418.298,Z 160.38,A -85,B 0,C 180,E1 -10276.736,E2 -10276.736} C_VEL
LIN {X 0,Y 418.289,Z 160.382,A -85,B 0,C 180,E1 -10279.803,E2 -10279.803} C_VEL
LIN {X 0,Y 418.23,Z 160.39,A -85,B 0,C 180,E1 -10282.737,E2 -10282.737} C_VEL
LIN {X 0,Y 418.224,Z 160.39,A -85,B 0,C 180,E1 -10285.907,E2 -10285.907} C_VEL
LIN {X 0,Y 418.247,Z 160.384,A -85,B 0,C 180,E1 -10289.163,E2 -10289.163} C_VEL
LIN {X 0,Y 418.245,Z 160.386,A -85,B 0,C 180,E1 -10292.845,E2 -10292.845} C_VEL
LIN {X 0,Y 418.237,Z 160.389,A -85,B 0,C 180,E1 -10296.24,E2 -10296.24} C_VEL
LIN {X 0,Y 418.244,Z 160.39,A -85,B 0,C 180,E1 -10299.683,E2 -10299.683} C_VEL
LIN {X 0,Y 418.221,Z 160.389,A -85,B 0,C 180,E1 -10302.323,E2 -10302.323} C_VEL
LIN {X 0,Y 418.232,Z 160.39,A -85,B 0,C 180,E1 -10305.111,E2 -10305.111} C_VEL
LIN {X 0,Y 418.233,Z 160.39,A -85,B 0,C 180,E1 -10307.769,E2 -10307.769} C_VEL
LIN {X 0,Y 418.239,Z 160.389,A -85,B 0,C 180,E1 -10311.559,E2 -10311.559} C_VEL
LIN {X 0,Y 418.251,Z 160.388,A -85,B 0,C 180,E1 -10315.161,E2 -10315.161} C_VEL
LIN {X 0,Y 418.24,Z 160.388,A -85,B 0,C 180,E1 -10317.474,E2 -10317.474} C_VEL
LIN {X 0,Y 418.271,Z 160.384,A -85,B 0,C 180,E1 -10320.895,E2 -10320.895} C_VEL
LIN {X 0,Y 418.256,Z 160.384,A -85,B 0,C 180,E1 -10324.097,E2 -10324.097} C_VEL
LIN {X 0,Y 418.233,Z 160.387,A -85,B 0,C 180,E1 -10327.266,E2 -10327.266} C_VEL
LIN {X 0,Y 418.281,Z 160.384,A -85,B 0,C 180,E1 -10330.366,E2 -10330.366} C_VEL
LIN {X 0,Y 418.315,Z 160.377,A -85,B 0,C 180,E1 -10333.406,E2 -10333.406} C_VEL
LIN {X 0,Y 418.345,Z 160.373,A -85,B 0,C 180,E1 -10337.001,E2 -10337.001} C_VEL
LIN {X 0,Y 418.339,Z 160.377,A -85,B 0,C 180,E1 -10340.33,E2 -10340.33} C_VEL
LIN {X 0,Y 418.513,Z 160.354,A -85,B 0,C 180,E1 -10342.281,E2 -10342.281} C_VEL
LIN {X 0,Y 418.514,Z 160.354,A -85,B 0,C 180,E1 -10344.219,E2 -10344.219} C_VEL
LIN {X 0,Y 418.543,Z 160.351,A -85,B 0,C 180,E1 -10348.077,E2 -10348.077} C_VEL
LIN {X 0,Y 418.544,Z 160.352,A -85,B 0,C 180,E1 -10350.002,E2 -10350.002} C_VEL
LIN {X 0,Y 418.495,Z 160.354,A -85,B 0,C 180,E1 -10352.889,E2 -10352.889} C_VEL
LIN {X 0,Y 418.497,Z 160.355,A -85,B 0,C 180,E1 -10356.752,E2 -10356.752} C_VEL
LIN {X 0,Y 418.359,Z 160.371,A -85,B 0,C 180,E1 -10359.165,E2 -10359.165} C_VEL
LIN {X 0,Y 418.359,Z 160.37,A -85,B 0,C 180,E1 -10362.616,E2 -10362.616} C_VEL
LIN {X 0,Y 418.324,Z 160.377,A -85,B 0,C 180,E1 -10363.355,E2 -10363.355} C_VEL
LIN {X 0,Y 417.63,Z 160.467,A -85,B 0,C 180,E1 -10364.158,E2 -10364.158} C_VEL
LIN {X 0,Y 414.752,Z 160.824,A -85,B 0,C 180,E1 -10365.464,E2 -10365.464} C_VEL
LIN {X 0,Y 412.34,Z 161.121,A -85,B 0,C 180,E1 -10366.518,E2 -10366.518} C_VEL
LIN {X 0,Y 411.319,Z 161.251,A -85,B 0,C 180,E1 -10367.333,E2 -10367.333} C_VEL
LIN {X 0,Y 411.243,Z 161.258,A -85,B 0,C 180,E1 -10367.609,E2 -10367.609} C_VEL
LIN {X 0,Y 411.201,Z 161.265,A -85,B 0,C 180,E1 -10371.035,E2 -10371.035} C_VEL
LIN {X 0,Y 411.196,Z 161.263,A -85,B 0,C 180,E1 -10374.219,E2 -10374.219} C_VEL
LIN {X 0,Y 411.153,Z 161.27,A -85,B 0,C 180,E1 -10377.487,E2 -10377.487} C_VEL
LIN {X 0,Y 411.201,Z 161.264,A -85,B 0,C 180,E1 -10379.714,E2 -10379.714} C_VEL
LIN {X 0,Y 411.211,Z 161.264,A -85,B 0,C 180,E1 -10383.157,E2 -10383.157} C_VEL
LIN {X 0,Y 411.194,Z 161.265,A -85,B 0,C 180,E1 -10386.553,E2 -10386.553} C_VEL
LIN {X 0,Y 411.172,Z 161.265,A -85,B 0,C 180,E1 -10389.721,E2 -10389.721} C_VEL
LIN {X 0,Y 411.17,Z 161.268,A -85,B 0,C 180,E1 -10393.135,E2 -10393.135} C_VEL
LIN {X 0,Y 411.173,Z 161.268,A -85,B 0,C 180,E1 -10395.882,E2 -10395.882} C_VEL
LIN {X 0,Y 411.167,Z 161.269,A -85,B 0,C 180,E1 -10398.773,E2 -10398.773} C_VEL
LIN {X 0,Y 411.188,Z 161.267,A -85,B 0,C 180,E1 -10402.026,E2 -10402.026} C_VEL
LIN {X 0,Y 411.215,Z 161.265,A -85,B 0,C 180,E1 -10405.667,E2 -10405.667} C_VEL
LIN {X 0,Y 411.285,Z 161.362,A -85,B 0,C 180,E1 -10407.005,E2 -10407.005} C_VEL
LIN {X 0,Y 412.082,Z 166.267,A -85,B 0,C 180,E1 -10409.226,E2 -10409.226} C_VEL
LIN {X 0,Y 411.98,Z 171.435,A -85,B 0,C 180,E1 -10411.468,E2 -10411.468} C_VEL
LIN {X 0,Y 411.613,Z 179.123,A -85,B 0,C 180,E1 -10414.732,E2 -10414.732} C_VEL
LIN {X 0,Y 411.205,Z 186.739,A -85,B 0,C 180,E1 -10417.913,E2 -10417.913} C_VEL
LIN {X 0,Y 410.948,Z 194.315,A -85,B 0,C 180,E1 -10421.038,E2 -10421.038} C_VEL
LIN {X 0,Y 410.656,Z 203.116,A -85,B 0,C 180,E1 -10424.617,E2 -10424.617} C_VEL
LIN {X 0,Y 410.408,Z 211.926,A -85,B 0,C 180,E1 -10428.142,E2 -10428.142} C_VEL
LIN {X 0,Y 410.315,Z 215.464,A -85,B 0,C 180,E1 -10429.546,E2 -10429.546} C_VEL
LIN {X 0,Y 411.592,Z 227.775,A -85,B 0,C 180,E1 -10430.231,E2 -10430.231} C_VEL
LIN {X 0,Y 411.803,Z 234.017,A -85,B 0,C 180,E1 -10430.669,E2 -10430.669} C_VEL
LIN {X 0,Y 411.376,Z 243.849,A -85,B 0,C 180,E1 -10431.527,E2 -10431.527} C_VEL
LIN {X 0,Y 411.089,Z 251.569,A -85,B 0,C 180,E1 -10432.396,E2 -10432.396} C_VEL
LIN {X 0,Y 410.817,Z 258.484,A -85,B 0,C 180,E1 -10433.369,E2 -10433.369} C_VEL
LIN {X 0,Y 410.576,Z 265.319,A -85,B 0,C 180,E1 -10434.598,E2 -10434.598} C_VEL
LIN {X 0,Y 410.447,Z 269.59,A -85,B 0,C 180,E1 -10435.581,E2 -10435.581} C_VEL
LIN {X 0,Y 410.256,Z 274.343,A -85,B 0,C 180,E1 -10437.054,E2 -10437.054} C_VEL
LIN {X 0,Y 410.1,Z 276.544,A -85,B 0,C 180,E1 -10438.036,E2 -10438.036} C_VEL
LIN {X 0,Y 410.046,Z 278.037,A -85,B 0,C 180,E1 -10439.018,E2 -10439.018} C_VEL
LIN {X 0,Y 410.053,Z 278.851,A -85,B 0,C 180,E1 -10440,E2 -10440} C_VEL
LIN {X 0,Y 410.133,Z 278.99,A -85,B 0,C 180,E1 -10440.982,E2 -10440.982} C_VEL
LIN {X 0,Y 410.268,Z 278.459,A -85,B 0,C 180,E1 -10441.963,E2 -10441.963} C_VEL
LIN {X 0,Y 410.477,Z 277.257,A -85,B 0,C 180,E1 -10442.944,E2 -10442.944} C_VEL
LIN {X 0,Y 410.778,Z 274.162,A -85,B 0,C 180,E1 -10444.416,E2 -10444.416} C_VEL
LIN {X 0,Y 410.919,Z 271.174,A -85,B 0,C 180,E1 -10445.398,E2 -10445.398} C_VEL
LIN {X 0,Y 411.247,Z 266.254,A -85,B 0,C 180,E1 -10446.624,E2 -10446.624} C_VEL
LIN {X 0,Y 411.743,Z 259.799,A -85,B 0,C 180,E1 -10447.848,E2 -10447.848} C_VEL
LIN {X 0,Y 412.51,Z 251.346,A -85,B 0,C 180,E1 -10449.067,E2 -10449.067} C_VEL
LIN {X 0,Y 413.18,Z 242.632,A -85,B 0,C 180,E1 -10450.041,E2 -10450.041} C_VEL
LIN {X 0,Y 413.669,Z 234.432,A -85,B 0,C 180,E1 -10450.771,E2 -10450.771} C_VEL
LIN {X 0,Y 412.44,Z 224.502,A -85,B 0,C 180,E1 -10451.55,E2 -10451.55} C_VEL
LIN {X 0,Y 410.816,Z 216.563,A -85,B 0,C 180,E1 -10452.102,E2 -10452.102} C_VEL
LIN {X 0,Y 411.209,Z 208.933,A -85,B 0,C 180,E1 -10455.362,E2 -10455.362} C_VEL
LIN {X 0,Y 411.615,Z 201.999,A -85,B 0,C 180,E1 -10458.414,E2 -10458.414} C_VEL
LIN {X 0,Y 412.167,Z 194.13,A -85,B 0,C 180,E1 -10462.032,E2 -10462.032} C_VEL
LIN {X 0,Y 412.853,Z 186.857,A -85,B 0,C 180,E1 -10465.547,E2 -10465.547} C_VEL
LIN {X 0,Y 413.78,Z 180.278,A -85,B 0,C 180,E1 -10468.952,E2 -10468.952} C_VEL
LIN {X 0,Y 414.017,Z 177.343,A -85,B 0,C 180,E1 -10470.614,E2 -10470.614} C_VEL
LIN {X 0,Y 414.009,Z 175.224,A -85,B 0,C 180,E1 -10471.92,E2 -10471.92} C_VEL
LIN {X 0,Y 413.537,Z 172.143,A -85,B 0,C 180,E1 -10474.113,E2 -10474.113} C_VEL
LIN {X 0,Y 412.91,Z 168.899,A -85,B 0,C 180,E1 -10476.871,E2 -10476.871} C_VEL
LIN {X 0,Y 412.506,Z 166.837,A -85,B 0,C 180,E1 -10479.078,E2 -10479.078} C_VEL
LIN {X 0,Y 412.12,Z 165.248,A -85,B 0,C 180,E1 -10481.689,E2 -10481.689} C_VEL
LIN {X 0,Y 411.994,Z 164.476,A -85,B 0,C 180,E1 -10484.379,E2 -10484.379} C_VEL
LIN {X 0,Y 412.062,Z 164.829,A -85,B 0,C 180,E1 -10487.172,E2 -10487.172} C_VEL
LIN {X 0,Y 412.46,Z 166.392,A -85,B 0,C 180,E1 -10490.065,E2 -10490.065} C_VEL
LIN {X 0,Y 412.934,Z 168.411,A -85,B 0,C 180,E1 -10492.213,E2 -10492.213} C_VEL
LIN {X 0,Y 413.727,Z 171.646,A -85,B 0,C 180,E1 -10494.72,E2 -10494.72} C_VEL
LIN {X 0,Y 414.615,Z 175.629,A -85,B 0,C 180,E1 -10497.15,E2 -10497.15} C_VEL
LIN {X 0,Y 415.601,Z 180.477,A -85,B 0,C 180,E1 -10499.591,E2 -10499.591} C_VEL
LIN {X 0,Y 416.241,Z 184.642,A -85,B 0,C 180,E1 -10501.401,E2 -10501.401} C_VEL
LIN {X 0,Y 415.767,Z 188.545,A -85,B 0,C 180,E1 -10502.844,E2 -10502.844} C_VEL
LIN {X 0,Y 414.161,Z 197.953,A -85,B 0,C 180,E1 -10505.966,E2 -10505.966} C_VEL
LIN {X 0,Y 412.75,Z 209.823,A -85,B 0,C 180,E1 -10509.624,E2 -10509.624} C_VEL
LIN {X 0,Y 411.795,Z 220.462,A -85,B 0,C 180,E1 -10512.682,E2 -10512.682} C_VEL
LIN {X 0,Y 413.937,Z 232.76,A -85,B 0,C 180,E1 -10513.201,E2 -10513.201} C_VEL
LIN {X 0,Y 414.625,Z 243.781,A -85,B 0,C 180,E1 -10513.758,E2 -10513.758} C_VEL
LIN {X 0,Y 413.976,Z 255.776,A -85,B 0,C 180,E1 -10514.49,E2 -10514.49} C_VEL
LIN {X 0,Y 413.1,Z 267.964,A -85,B 0,C 180,E1 -10515.466,E2 -10515.466} C_VEL
LIN {X 0,Y 412.313,Z 277.98,A -85,B 0,C 180,E1 -10516.477,E2 -10516.477} C_VEL
LIN {X 0,Y 411.74,Z 287.539,A -85,B 0,C 180,E1 -10517.679,E2 -10517.679} C_VEL
LIN {X 0,Y 411.129,Z 295.611,A -85,B 0,C 180,E1 -10518.911,E2 -10518.911} C_VEL
LIN {X 0,Y 410.609,Z 303.513,A -85,B 0,C 180,E1 -10520.392,E2 -10520.392} C_VEL
LIN {X 0,Y 410.258,Z 310.725,A -85,B 0,C 180,E1 -10522.122,E2 -10522.122} C_VEL
LIN {X 0,Y 410.044,Z 315.991,A -85,B 0,C 180,E1 -10523.775,E2 -10523.775} C_VEL
LIN {X 0,Y 410.054,Z 319.146,A -85,B 0,C 180,E1 -10525.082,E2 -10525.082} C_VEL
LIN {X 0,Y 409.966,Z 320.956,A -85,B 0,C 180,E1 -10526.067,E2 -10526.067} C_VEL
LIN {X 0,Y 410.02,Z 322.337,A -85,B 0,C 180,E1 -10527.051,E2 -10527.051} C_VEL
LIN {X 0,Y 410.041,Z 323.305,A -85,B 0,C 180,E1 -10528.034,E2 -10528.034} C_VEL
LIN {X 0,Y 410.006,Z 323.81,A -85,B 0,C 180,E1 -10529.016,E2 -10529.016} C_VEL
LIN {X 0,Y 410.04,Z 323.893,A -85,B 0,C 180,E1 -10529.998,E2 -10529.998} C_VEL
LIN {X 0,Y 410.041,Z 323.571,A -85,B 0,C 180,E1 -10530.981,E2 -10530.981} C_VEL
LIN {X 0,Y 410.06,Z 322.804,A -85,B 0,C 180,E1 -10531.963,E2 -10531.963} C_VEL
LIN {X 0,Y 410.089,Z 321.587,A -85,B 0,C 180,E1 -10532.945,E2 -10532.945} C_VEL
LIN {X 0,Y 410.019,Z 318.916,A -85,B 0,C 180,E1 -10534.422,E2 -10534.422} C_VEL
LIN {X 0,Y 410.049,Z 315.153,A -85,B 0,C 180,E1 -10535.901,E2 -10535.901} C_VEL
LIN {X 0,Y 410.181,Z 310.194,A -85,B 0,C 180,E1 -10537.382,E2 -10537.382} C_VEL
LIN {X 0,Y 410.364,Z 303.858,A -85,B 0,C 180,E1 -10538.865,E2 -10538.865} C_VEL
LIN {X 0,Y 410.696,Z 295.821,A -85,B 0,C 180,E1 -10540.349,E2 -10540.349} C_VEL
LIN {X 0,Y 411.205,Z 287.581,A -85,B 0,C 180,E1 -10541.583,E2 -10541.583} C_VEL
LIN {X 0,Y 411.706,Z 278.533,A -85,B 0,C 180,E1 -10542.694,E2 -10542.694} C_VEL
LIN {X 0,Y 412.182,Z 267.191,A -85,B 0,C 180,E1 -10543.809,E2 -10543.809} C_VEL
LIN {X 0,Y 412.772,Z 256.086,A -85,B 0,C 180,E1 -10544.669,E2 -10544.669} C_VEL
LIN {X 0,Y 413.276,Z 243.493,A -85,B 0,C 180,E1 -10545.407,E2 -10545.407} C_VEL
LIN {X 0,Y 412.838,Z 235.785,A -85,B 0,C 180,E1 -10545.772,E2 -10545.772} C_VEL
LIN {X 0,Y 411.426,Z 222.897,A -85,B 0,C 180,E1 -10546.226,E2 -10546.226} C_VEL
LIN {X 0,Y 411.19,Z 220.332,A -85,B 0,C 180,E1 -10546.315,E2 -10546.315} C_VEL
LIN {X 0,Y 412.026,Z 206.791,A -85,B 0,C 180,E1 -10549.945,E2 -10549.945} C_VEL
LIN {X 0,Y 413.091,Z 193.383,A -85,B 0,C 180,E1 -10553.596,E2 -10553.596} C_VEL
LIN {X 0,Y 414.294,Z 180.171,A -85,B 0,C 180,E1 -10557.257,E2 -10557.257} C_VEL
LIN {X 0,Y 414.174,Z 176.354,A -85,B 0,C 180,E1 -10558.365,E2 -10558.365} C_VEL
LIN {X 0,Y 412.135,Z 166.144,A -85,B 0,C 180,E1 -10561.5,E2 -10561.5} C_VEL
LIN {X 0,Y 411.195,Z 161.267,A -85,B 0,C 180,E1 -10563.096,E2 -10563.096} C_VEL
LIN {X 0,Y 411.193,Z 161.27,A -85,B 0,C 180,E1 -10565.527,E2 -10565.527} C_VEL
LIN {X 0,Y 411.202,Z 161.264,A -85,B 0,C 180,E1 -10569.223,E2 -10569.223} C_VEL
LIN {X 0,Y 411.169,Z 161.27,A -85,B 0,C 180,E1 -10572.694,E2 -10572.694} C_VEL
LIN {X 0,Y 411.227,Z 161.261,A -85,B 0,C 180,E1 -10575.87,E2 -10575.87} C_VEL
LIN {X 0,Y 411.201,Z 161.266,A -85,B 0,C 180,E1 -10578.763,E2 -10578.763} C_VEL
LIN {X 0,Y 411.188,Z 161.266,A -85,B 0,C 180,E1 -10582.025,E2 -10582.025} C_VEL
LIN {X 0,Y 411.194,Z 161.264,A -85,B 0,C 180,E1 -10585.665,E2 -10585.665} C_VEL
LIN {X 0,Y 411.186,Z 161.265,A -85,B 0,C 180,E1 -10589.152,E2 -10589.152} C_VEL
LIN {X 0,Y 411.247,Z 161.259,A -85,B 0,C 180,E1 -10592.521,E2 -10592.521} C_VEL
